LIN {X 0,Y 411.273,Z 176.254,A -85,B 0,C 180,E1 -10451.833,E2 -10451.833} C_VEL
LIN {X 0,Y 411.231,Z 176.261,A -85,B 0,C 180,E1 -10454.854,E2 -10454.854} C_VEL
LIN {X 0,Y 411.22,Z 176.261,A -85,B 0,C 180,E1 -10457.916,E2 -10457.916} C_VEL
LIN {X 0,Y 411.208,Z 176.265,A -85,B 0,C 180,E1 -10461.033,E2 -10461.033} C_VEL
LIN {X 0,Y 411.202,Z 176.262,A -85,B 0,C 180,E1 -10464.217,E2 -10464.217} C_VEL
LIN {X 0,Y 411.232,Z 176.258,A -85,B 0,C 180,E1 -10467.48,E2 -10467.48} C_VEL
LIN {X 0,Y 411.171,Z 176.269,A -85,B 0,C 180,E1 -10470.849,E2 -10470.849} C_VEL
LIN {X 0,Y 411.181,Z 176.268,A -85,B 0,C 180,E1 -10474.336,E2 -10474.336} C_VEL
LIN {X 0,Y 411.182,Z 176.266,A -85,B 0,C 180,E1 -10477.975,E2 -10477.975} C_VEL
LIN {X 0,Y 411.189,Z 176.264,A -85,B 0,C 180,E1 -10481.238,E2 -10481.238} C_VEL
LIN {X 0,Y 411.214,Z 176.264,A -85,B 0,C 180,E1 -10484.485,E2 -10484.485} C_VEL
LIN {X 0,Y 411.208,Z 176.268,A -85,B 0,C 180,E1 -10487.3,E2 -10487.3} C_VEL
LIN {X 0,Y 411.201,Z 176.348,A -85,B 0,C 180,E1 -10489.503,E2 -10489.503} C_VEL
LIN {X 0,Y 411.973,Z 180.687,A -85,B 0,C 180,E1 -10492.115,E2 -10492.115} C_VEL
LIN {X 0,Y 412.375,Z 185.022,A -85,B 0,C 180,E1 -10494.592,E2 -10494.592} C_VEL
LIN {X 0,Y 411.962,Z 191.551,A -85,B 0,C 180,E1 -10498.075,E2 -10498.075} C_VEL
LIN {X 0,Y 411.48,Z 198.091,A -85,B 0,C 180,E1 -10501.433,E2 -10501.433} C_VEL
LIN {X 0,Y 411.07,Z 205.195,A -85,B 0,C 180,E1 -10504.977,E2 -10504.977} C_VEL
LIN {X 0,Y 410.743,Z 212.225,A -85,B 0,C 180,E1 -10508.418,E2 -10508.418} C_VEL
LIN {X 0,Y 410.41,Z 219.753,A -85,B 0,C 180,E1 -10512.049,E2 -10512.049} C_VEL
LIN {X 0,Y 410.348,Z 220.824,A -85,B 0,C 180,E1 -10512.562,E2 -10512.562} C_VEL
LIN {X 0,Y 412.666,Z 234.125,A -85,B 0,C 180,E1 -10513.061,E2 -10513.061} C_VEL
LIN {X 0,Y 414.357,Z 246.561,A -85,B 0,C 180,E1 -10513.709,E2 -10513.709} C_VEL
LIN {X 0,Y 414.471,Z 252.147,A -85,B 0,C 180,E1 -10514.042,E2 -10514.042} C_VEL
LIN {X 0,Y 413.707,Z 263.943,A -85,B 0,C 180,E1 -10514.861,E2 -10514.861} C_VEL
LIN {X 0,Y 412.966,Z 274.206,A -85,B 0,C 180,E1 -10515.766,E2 -10515.766} C_VEL
LIN {X 0,Y 412.217,Z 284.881,A -85,B 0,C 180,E1 -10516.946,E2 -10516.946} C_VEL
LIN {X 0,Y 411.604,Z 293.906,A -85,B 0,C 180,E1 -10518.178,E2 -10518.178} C_VEL
LIN {X 0,Y 410.954,Z 302.716,A -85,B 0,C 180,E1 -10519.657,E2 -10519.657} C_VEL
LIN {X 0,Y 410.528,Z 309.753,A -85,B 0,C 180,E1 -10521.138,E2 -10521.138} C_VEL
LIN {X 0,Y 410.19,Z 315.381,A -85,B 0,C 180,E1 -10522.618,E2 -10522.618} C_VEL
LIN {X 0,Y 410.035,Z 319.809,A -85,B 0,C 180,E1 -10524.098,E2 -10524.098} C_VEL
LIN {X 0,Y 410.019,Z 322.149,A -85,B 0,C 180,E1 -10525.085,E2 -10525.085} C_VEL
LIN {X 0,Y 409.932,Z 324.056,A -85,B 0,C 180,E1 -10526.069,E2 -10526.069} C_VEL
LIN {X 0,Y 409.926,Z 325.518,A -85,B 0,C 180,E1 -10527.053,E2 -10527.053} C_VEL
LIN {X 0,Y 409.966,Z 326.551,A -85,B 0,C 180,E1 -10528.036,E2 -10528.036} C_VEL
LIN {X 0,Y 409.927,Z 327.448,A -85,B 0,C 180,E1 -10530.001,E2 -10530.001} C_VEL
LIN {X 0,Y 409.935,Z 327.293,A -85,B 0,C 180,E1 -10530.983,E2 -10530.983} C_VEL
LIN {X 0,Y 409.966,Z 326.72,A -85,B 0,C 180,E1 -10531.965,E2 -10531.965} C_VEL
LIN {X 0,Y 409.931,Z 324.402,A -85,B 0,C 180,E1 -10533.933,E2 -10533.933} C_VEL
LIN {X 0,Y 410.018,Z 321.536,A -85,B 0,C 180,E1 -10535.41,E2 -10535.41} C_VEL
LIN {X 0,Y 410.168,Z 317.645,A -85,B 0,C 180,E1 -10536.889,E2 -10536.889} C_VEL
LIN {X 0,Y 410.421,Z 312.629,A -85,B 0,C 180,E1 -10538.369,E2 -10538.369} C_VEL
LIN {X 0,Y 410.84,Z 306.335,A -85,B 0,C 180,E1 -10539.85,E2 -10539.85} C_VEL
LIN {X 0,Y 411.402,Z 298.458,A -85,B 0,C 180,E1 -10541.33,E2 -10541.33} C_VEL
LIN {X 0,Y 412.128,Z 290.44,A -85,B 0,C 180,E1 -10542.558,E2 -10542.558} C_VEL
LIN {X 0,Y 412.802,Z 280.664,A -85,B 0,C 180,E1 -10543.789,E2 -10543.789} C_VEL
LIN {X 0,Y 413.655,Z 269.786,A -85,B 0,C 180,E1 -10544.89,E2 -10544.89} C_VEL
LIN {X 0,Y 414.435,Z 259.142,A -85,B 0,C 180,E1 -10545.743,E2 -10545.743} C_VEL
LIN {X 0,Y 414.947,Z 248.593,A -85,B 0,C 180,E1 -10546.417,E2 -10546.417} C_VEL
LIN {X 0,Y 413.347,Z 236.158,A -85,B 0,C 180,E1 -10547.103,E2 -10547.103} C_VEL
LIN {X 0,Y 410.794,Z 222.945,A -85,B 0,C 180,E1 -10547.664,E2 -10547.664} C_VEL
LIN {X 0,Y 410.406,Z 220.684,A -85,B 0,C 180,E1 -10547.759,E2 -10547.759} C_VEL
LIN {X 0,Y 410.738,Z 213.884,A -85,B 0,C 180,E1 -10551.058,E2 -10551.058} C_VEL
LIN {X 0,Y 411.04,Z 207.48,A -85,B 0,C 180,E1 -10554.226,E2 -10554.226} C_VEL
LIN {X 0,Y 411.432,Z 201.028,A -85,B 0,C 180,E1 -10557.464,E2 -10557.464} C_VEL
LIN {X 0,Y 411.887,Z 194.581,A -85,B 0,C 180,E1 -10560.788,E2 -10560.788} C_VEL
LIN {X 0,Y 412.246,Z 189.772,A -85,B 0,C 180,E1 -10563.347,E2 -10563.347} C_VEL
LIN {X 0,Y 412.463,Z 184.976,A -85,B 0,C 180,E1 -10566.002,E2 -10566.002} C_VEL
LIN {X 0,Y 412.038,Z 181.046,A -85,B 0,C 180,E1 -10568.316,E2 -10568.316} C_VEL
LIN {X 0,Y 411.221,Z 176.262,A -85,B 0,C 180,E1 -10571.317,E2 -10571.317} C_VEL
LIN {X 0,Y 411.217,Z 176.263,A -85,B 0,C 180,E1 -10574.482,E2 -10574.482} C_VEL
LIN {X 0,Y 411.163,Z 176.268,A -85,B 0,C 180,E1 -10578.193,E2 -10578.193} C_VEL
LIN {X 0,Y 411.193,Z 176.264,A -85,B 0,C 180,E1 -10580.773,E2 -10580.773} C_VEL
LIN {X 0,Y 411.181,Z 176.264,A -85,B 0,C 180,E1 -10584.47,E2 -10584.47} C_VEL
LIN {X 0,Y 411.19,Z 176.265,A -85,B 0,C 180,E1 -10586.872,E2 -10586.872} C_VEL
LIN {X 0,Y 411.196,Z 176.264,A -85,B 0,C 180,E1 -10590.647,E2 -10590.647} C_VEL
LIN {X 0,Y 411.218,Z 176.261,A -85,B 0,C 180,E1 -10593.618,E2 -10593.618} C_VEL
LIN {X 0,Y 411.236,Z 176.259,A -85,B 0,C 180,E1 -10597.339,E2 -10597.339} C_VEL
LIN {X 0,Y 411.244,Z 176.256,A -85,B 0,C 180,E1 -10600.03,E2 -10600.03} C_VEL
LIN {X 0,Y 411.242,Z 176.26,A -85,B 0,C 180,E1 -10603.13,E2 -10603.13} C_VEL
LIN {X 0,Y 411.289,Z 176.255,A -85,B 0,C 180,E1 -10606.891,E2 -10606.891} C_VEL
LIN {X 0,Y 411.288,Z 176.253,A -85,B 0,C 180,E1 -10610.161,E2 -10610.161} C_VEL
LIN {X 0,Y 411.457,Z 176.23,A -85,B 0,C 180,E1 -10613.133,E2 -10613.133} C_VEL
LIN {X 0,Y 411.296,Z 176.251,A -85,B 0,C 180,E1 -10615.099,E2 -10615.099} C_VEL
LIN {X 0,Y 411.484,Z 176.231,A -85,B 0,C 180,E1 -10618.043,E2 -10618.043} C_VEL
LIN {X 0,Y 411.611,Z 176.214,A -85,B 0,C 180,E1 -10620,E2 -10620} C_VEL
LIN {X 0,Y 411.451,Z 176.23,A -85,B 0,C 180,E1 -10622.938,E2 -10622.938} C_VEL
LIN {X 0,Y 411.431,Z 176.233,A -85,B 0,C 180,E1 -10626.604,E2 -10626.604} C_VEL
LIN {X 0,Y 411.268,Z 176.258,A -85,B 0,C 180,E1 -10629.84,E2 -10629.84} C_VEL
LIN {X 0,Y 411.282,Z 176.253,A -85,B 0,C 180,E1 -10633.104,E2 -10633.104} C_VEL
LIN {X 0,Y 411.281,Z 176.251,A -85,B 0,C 180,E1 -10636.888,E2 -10636.888} C_VEL
LIN {X 0,Y 411.21,Z 176.263,A -85,B 0,C 180,E1 -10639.988,E2 -10639.988} C_VEL
LIN {X 0,Y 411.183,Z 176.268,A -85,B 0,C 180,E1 -10643.149,E2 -10643.149} C_VEL
LIN {X 0,Y 411.219,Z 176.259,A -85,B 0,C 180,E1 -10646.383,E2 -10646.383} C_VEL
LIN {X 0,Y 411.193,Z 176.264,A -85,B 0,C 180,E1 -10649.714,E2 -10649.714} C_VEL
LIN {X 0,Y 411.191,Z 176.267,A -85,B 0,C 180,E1 -10653.158,E2 -10653.158} C_VEL
LIN {X 0,Y 411.178,Z 176.267,A -85,B 0,C 180,E1 -10656.554,E2 -10656.554} C_VEL
LIN {X 0,Y 411.196,Z 176.262,A -85,B 0,C 180,E1 -10659.729,E2 -10659.729} C_VEL
LIN {X 0,Y 411.162,Z 176.269,A -85,B 0,C 180,E1 -10663.136,E2 -10663.136} C_VEL
LIN {X 0,Y 411.159,Z 176.267,A -85,B 0,C 180,E1 -10665.883,E2 -10665.883} C_VEL
LIN {X 0,Y 411.154,Z 176.272,A -85,B 0,C 180,E1 -10668.774,E2 -10668.774} C_VEL
LIN {X 0,Y 411.093,Z 176.295,A -85,B 0,C 180,E1 -10671.852,E2 -10671.852} C_VEL
LIN {X 0,Y 411.092,Z 179.421,A -85,B 0,C 180,E1 -10674.463,E2 -10674.463} C_VEL
LIN {X 0,Y 410.927,Z 183.802,A -85,B 0,C 180,E1 -10677.984,E2 -10677.984} C_VEL
LIN {X 0,Y 410.72,Z 188.143,A -85,B 0,C 180,E1 -10681.374,E2 -10681.374} C_VEL
LIN {X 0,Y 410.555,Z 192.532,A -85,B 0,C 180,E1 -10684.663,E2 -10684.663} C_VEL
LIN {X 0,Y 410.421,Z 196.937,A -85,B 0,C 180,E1 -10687.87,E2 -10687.87} C_VEL
LIN {X 0,Y 410.363,Z 200.38,A -85,B 0,C 180,E1 -10690.327,E2 -10690.327} C_VEL
LIN {X 0,Y 413.785,Z 215.04,A -85,B 0,C 180,E1 -10690.995,E2 -10690.995} C_VEL
LIN {X 0,Y 415.59,Z 225.146,A -85,B 0,C 180,E1 -10691.579,E2 -10691.579} C_VEL
LIN {X 0,Y 414.916,Z 237.745,A -85,B 0,C 180,E1 -10692.376,E2 -10692.376} C_VEL
LIN {X 0,Y 414.043,Z 249.487,A -85,B 0,C 180,E1 -10693.356,E2 -10693.356} C_VEL
LIN {X 0,Y 413.36,Z 258.933,A -85,B 0,C 180,E1 -10694.342,E2 -10694.342} C_VEL
LIN {X 0,Y 412.494,Z 269.466,A -85,B 0,C 180,E1 -10695.697,E2 -10695.697} C_VEL
LIN {X 0,Y 411.837,Z 277.292,A -85,B 0,C 180,E1 -10696.949,E2 -10696.949} C_VEL
LIN {X 0,Y 411.318,Z 284.751,A -85,B 0,C 180,E1 -10698.418,E2 -10698.418} C_VEL
LIN {X 0,Y 410.81,Z 289.915,A -85,B 0,C 180,E1 -10699.652,E2 -10699.652} C_VEL
LIN {X 0,Y 410.499,Z 294.904,A -85,B 0,C 180,E1 -10701.136,E2 -10701.136} C_VEL
LIN {X 0,Y 410.23,Z 298.768,A -85,B 0,C 180,E1 -10702.618,E2 -10702.618} C_VEL
LIN {X 0,Y 410.073,Z 301.606,A -85,B 0,C 180,E1 -10704.098,E2 -10704.098} C_VEL
LIN {X 0,Y 410.043,Z 302.944,A -85,B 0,C 180,E1 -10705.084,E2 -10705.084} C_VEL
LIN {X 0,Y 409.969,Z 304.457,A -85,B 0,C 180,E1 -10707.052,E2 -10707.052} C_VEL
LIN {X 0,Y 410.003,Z 304.609,A -85,B 0,C 180,E1 -10708.035,E2 -10708.035} C_VEL
LIN {X 0,Y 409.931,Z 303.724,A -85,B 0,C 180,E1 -10709.999,E2 -10709.999} C_VEL
LIN {X 0,Y 409.97,Z 302.708,A -85,B 0,C 180,E1 -10710.982,E2 -10710.982} C_VEL
LIN {X 0,Y 410.076,Z 301.27,A -85,B 0,C 180,E1 -10711.963,E2 -10711.963} C_VEL
LIN {X 0,Y 410.309,Z 298.319,A -85,B 0,C 180,E1 -10713.436,E2 -10713.436} C_VEL
LIN {X 0,Y 410.422,Z 294.338,A -85,B 0,C 180,E1 -10714.911,E2 -10714.911} C_VEL
LIN {X 0,Y 410.865,Z 288.202,A -85,B 0,C 180,E1 -10716.629,E2 -10716.629} C_VEL
LIN {X 0,Y 411.324,Z 281.524,A -85,B 0,C 180,E1 -10718.102,E2 -10718.102} C_VEL
LIN {X 0,Y 411.935,Z 273.234,A -85,B 0,C 180,E1 -10719.574,E2 -10719.574} C_VEL
LIN {X 0,Y 412.14,Z 271.122,A -85,B 0,C 180,E1 -10719.894,E2 -10719.894} C_VEL
LIN {X 0,Y 411.831,Z 267.118,A -85,B 0,C 180,E1 -10720.493,E2 -10720.493} C_VEL
LIN {X 0,Y 409.616,Z 260.349,A -85,B 0,C 180,E1 -10721.45,E2 -10721.45} C_VEL
LIN {X 0,Y 407.273,Z 253.153,A -85,B 0,C 180,E1 -10722.35,E2 -10722.35} C_VEL
LIN {X 0,Y 406.767,Z 248.372,A -85,B 0,C 180,E1 -10722.849,E2 -10722.849} C_VEL
LIN {X 0,Y 407.614,Z 237.96,A -85,B 0,C 180,E1 -10723.712,E2 -10723.712} C_VEL
LIN {X 0,Y 408.173,Z 227.39,A -85,B 0,C 180,E1 -10724.411,E2 -10724.411} C_VEL
LIN {X 0,Y 408.052,Z 223.747,A -85,B 0,C 180,E1 -10724.624,E2 -10724.624} C_VEL
LIN {X 0,Y 405.676,Z 211.271,A -85,B 0,C 180,E1 -10725.307,E2 -10725.307} C_VEL
LIN {X 0,Y 403.286,Z 200.508,A -85,B 0,C 180,E1 -10725.767,E2 -10725.767} C_VEL
LIN {X 0,Y 403.368,Z 195.566,A -85,B 0,C 180,E1 -10729.33,E2 -10729.33} C_VEL
LIN {X 0,Y 403.532,Z 191.072,A -85,B 0,C 180,E1 -10732.621,E2 -10732.621} C_VEL
LIN {X 0,Y 403.664,Z 186.904,A -85,B 0,C 180,E1 -10735.799,E2 -10735.799} C_VEL
LIN {X 0,Y 403.861,Z 182.638,A -85,B 0,C 180,E1 -10739.157,E2 -10739.157} C_VEL
LIN {X 0,Y 403.988,Z 179.68,A -85,B 0,C 180,E1 -10741.522,E2 -10741.522} C_VEL
LIN {X 0,Y 403.986,Z 177.43,A -85,B 0,C 180,E1 -10743.379,E2 -10743.379} C_VEL
LIN {X 0,Y 404.088,Z 177.151,A -85,B 0,C 180,E1 -10745.17,E2 -10745.17} C_VEL
LIN {X 0,Y 404.136,Z 177.142,A -85,B 0,C 180,E1 -10748.504,E2 -10748.504} C_VEL
LIN {X 0,Y 404.11,Z 177.149,A -85,B 0,C 180,E1 -10751.597,E2 -10751.597} C_VEL
LIN {X 0,Y 404.141,Z 177.142,A -85,B 0,C 180,E1 -10754.521,E2 -10754.521} C_VEL
LIN {X 0,Y 404.189,Z 177.139,A -85,B 0,C 180,E1 -10757.302,E2 -10757.302} C_VEL
LIN {X 0,Y 404.15,Z 177.14,A -85,B 0,C 180,E1 -10759.953,E2 -10759.953} C_VEL
LIN {X 0,Y 404.116,Z 177.148,A -85,B 0,C 180,E1 -10763.122,E2 -10763.122} C_VEL
LIN {X 0,Y 404.122,Z 177.145,A -85,B 0,C 180,E1 -10766.185,E2 -10766.185} C_VEL
LIN {X 0,Y 404.128,Z 177.143,A -85,B 0,C 180,E1 -10769.713,E2 -10769.713} C_VEL
LIN {X 0,Y 404.17,Z 177.139,A -85,B 0,C 180,E1 -10773.121,E2 -10773.121} C_VEL
LIN {X 0,Y 404.154,Z 177.144,A -85,B 0,C 180,E1 -10776.424,E2 -10776.424} C_VEL
LIN {X 0,Y 404.198,Z 177.136,A -85,B 0,C 180,E1 -10779.859,E2 -10779.859} C_VEL
LIN {X 0,Y 404.188,Z 177.137,A -85,B 0,C 180,E1 -10782.99,E2 -10782.99} C_VEL
LIN {X 0,Y 404.197,Z 177.138,A -85,B 0,C 180,E1 -10785.911,E2 -10785.911} C_VEL
LIN {X 0,Y 404.254,Z 177.127,A -85,B 0,C 180,E1 -10788.975,E2 -10788.975} C_VEL
LIN {X 0,Y 404.402,Z 177.113,A -85,B 0,C 180,E1 -10792.097,E2 -10792.097} C_VEL
LIN {X 0,Y 404.418,Z 177.111,A -85,B 0,C 180,E1 -10794.015,E2 -10794.015} C_VEL
LIN {X 0,Y 404.447,Z 177.107,A -85,B 0,C 180,E1 -10798.008,E2 -10798.008} C_VEL
LIN {X 0,Y 404.574,Z 177.091,A -85,B 0,C 180,E1 -10800,E2 -10800} C_VEL
LIN {X 0,Y 404.4,Z 177.11,A -85,B 0,C 180,E1 -10802.988,E2 -10802.988} C_VEL
LIN {X 0,Y 404.409,Z 177.11,A -85,B 0,C 180,E1 -10805.985,E2 -10805.985} C_VEL
LIN {X 0,Y 404.289,Z 177.124,A -85,B 0,C 180,E1 -10809.001,E2 -10809.001} C_VEL
LIN {X 0,Y 404.242,Z 177.129,A -85,B 0,C 180,E1 -10812.042,E2 -10812.042} C_VEL
LIN {X 0,Y 404.176,Z 177.142,A -85,B 0,C 180,E1 -10815.119,E2 -10815.119} C_VEL
LIN {X 0,Y 404.181,Z 177.137,A -85,B 0,C 180,E1 -10818.239,E2 -10818.239} C_VEL
LIN {X 0,Y 404.164,Z 177.142,A -85,B 0,C 180,E1 -10821.418,E2 -10821.418} C_VEL
LIN {X 0,Y 404.151,Z 177.143,A -85,B 0,C 180,E1 -10824.667,E2 -10824.667} C_VEL
LIN {X 0,Y 404.17,Z 177.137,A -85,B 0,C 180,E1 -10828.001,E2 -10828.001} C_VEL
LIN {X 0,Y 404.116,Z 177.145,A -85,B 0,C 180,E1 -10831.561,E2 -10831.561} C_VEL
LIN {X 0,Y 404.161,Z 177.142,A -85,B 0,C 180,E1 -10835.018,E2 -10835.018} C_VEL
LIN {X 0,Y 404.142,Z 177.145,A -85,B 0,C 180,E1 -10838.758,E2 -10838.758} C_VEL
LIN {X 0,Y 404.171,Z 177.138,A -85,B 0,C 180,E1 -10841.613,E2 -10841.613} C_VEL
LIN {X 0,Y 404.179,Z 177.14,A -85,B 0,C 180,E1 -10844.532,E2 -10844.532} C_VEL
LIN {X 0,Y 404.187,Z 177.143,A -85,B 0,C 180,E1 -10847.307,E2 -10847.307} C_VEL
LIN {X 0,Y 404.187,Z 177.286,A -85,B 0,C 180,E1 -10849.309,E2 -10849.309} C_VEL
LIN {X 0,Y 404.938,Z 181.679,A -85,B 0,C 180,E1 -10852.001,E2 -10852.001} C_VEL
LIN {X 0,Y 405.354,Z 186.104,A -85,B 0,C 180,E1 -10854.576,E2 -10854.576} C_VEL
LIN {X 0,Y 404.913,Z 192.898,A -85,B 0,C 180,E1 -10858.264,E2 -10858.264} C_VEL
LIN {X 0,Y 404.428,Z 199.01,A -85,B 0,C 180,E1 -10861.456,E2 -10861.456} C_VEL
LIN {X 0,Y 404.048,Z 205.484,A -85,B 0,C 180,E1 -10864.754,E2 -10864.754} C_VEL
LIN {X 0,Y 403.652,Z 213.104,A -85,B 0,C 180,E1 -10868.556,E2 -10868.556} C_VEL
LIN {X 0,Y 403.301,Z 220.736,A -85,B 0,C 180,E1 -10872.265,E2 -10872.265} C_VEL
LIN {X 0,Y 405.694,Z 234.188,A -85,B 0,C 180,E1 -10872.787,E2 -10872.787} C_VEL
LIN {X 0,Y 407.406,Z 246.932,A -85,B 0,C 180,E1 -10873.47,E2 -10873.47} C_VEL
LIN {X 0,Y 407.615,Z 252.022,A -85,B 0,C 180,E1 -10873.784,E2 -10873.784} C_VEL
LIN {X 0,Y 406.827,Z 263.573,A -85,B 0,C 180,E1 -10874.599,E2 -10874.599} C_VEL
LIN {X 0,Y 405.996,Z 274.629,A -85,B 0,C 180,E1 -10875.593,E2 -10875.593} C_VEL
LIN {X 0,Y 405.276,Z 284.759,A -85,B 0,C 180,E1 -10876.742,E2 -10876.742} C_VEL
LIN {X 0,Y 404.622,Z 293.619,A -85,B 0,C 180,E1 -10877.971,E2 -10877.971} C_VEL
LIN {X 0,Y 403.918,Z 302.445,A -85,B 0,C 180,E1 -10879.475,E2 -10879.475} C_VEL
LIN {X 0,Y 403.483,Z 309.501,A -85,B 0,C 180,E1 -10880.982,E2 -10880.982} C_VEL
LIN {X 0,Y 403.137,Z 315.141,A -85,B 0,C 180,E1 -10882.488,E2 -10882.488} C_VEL
LIN {X 0,Y 402.966,Z 319.578,A -85,B 0,C 180,E1 -10883.994,E2 -10883.994} C_VEL
LIN {X 0,Y 402.932,Z 321.923,A -85,B 0,C 180,E1 -10884.998,E2 -10884.998} C_VEL
LIN {X 0,Y 402.852,Z 323.835,A -85,B 0,C 180,E1 -10885.999,E2 -10885.999} C_VEL
LIN {X 0,Y 402.825,Z 325.305,A -85,B 0,C 180,E1 -10887.001,E2 -10887.001} C_VEL
LIN {X 0,Y 402.864,Z 326.342,A -85,B 0,C 180,E1 -10888.001,E2 -10888.001} C_VEL
LIN {X 0,Y 402.862,Z 326.989,A -85,B 0,C 180,E1 -10889.001,E2 -10889.001} C_VEL
LIN {X 0,Y 402.851,Z 327.249,A -85,B 0,C 180,E1 -10890.001,E2 -10890.001} C_VEL
LIN {X 0,Y 402.862,Z 327.103,A -85,B 0,C 180,E1 -10891,E2 -10891} C_VEL
LIN {X 0,Y 402.864,Z 326.533,A -85,B 0,C 180,E1 -10892,E2 -10892} C_VEL
LIN {X 0,Y 402.852,Z 324.223,A -85,B 0,C 180,E1 -10894.002,E2 -10894.002} C_VEL
LIN {X 0,Y 402.916,Z 321.366,A -85,B 0,C 180,E1 -10895.505,E2 -10895.505} C_VEL
LIN {X 0,Y 403.082,Z 317.484,A -85,B 0,C 180,E1 -10897.011,E2 -10897.011} C_VEL
LIN {X 0,Y 403.363,Z 312.478,A -85,B 0,C 180,E1 -10898.517,E2 -10898.517} C_VEL
LIN {X 0,Y 403.829,Z 306.197,A -85,B 0,C 180,E1 -10900.022,E2 -10900.022} C_VEL
LIN {X 0,Y 404.417,Z 298.339,A -85,B 0,C 180,E1 -10901.528,E2 -10901.528} C_VEL
LIN {X 0,Y 405.173,Z 290.338,A -85,B 0,C 180,E1 -10902.777,E2 -10902.777} C_VEL
LIN {X 0,Y 405.871,Z 280.581,A -85,B 0,C 180,E1 -10904.029,E2 -10904.029} C_VEL
LIN {X 0,Y 406.791,Z 269.735,A -85,B 0,C 180,E1 -10905.147,E2 -10905.147} C_VEL
LIN {X 0,Y 407.604,Z 259.135,A -85,B 0,C 180,E1 -10906.014,E2 -10906.014} C_VEL
LIN {X 0,Y 408.152,Z 249.946,A -85,B 0,C 180,E1 -10906.621,E2 -10906.621} C_VEL
LIN {X 0,Y 406.835,Z 238.963,A -85,B 0,C 180,E1 -10907.269,E2 -10907.269} C_VEL
LIN {X 0,Y 404.358,Z 225.626,A -85,B 0,C 180,E1 -10907.886,E2 -10907.886} C_VEL
LIN {X 0,Y 403.357,Z 220.523,A -85,B 0,C 180,E1 -10908.08,E2 -10908.08} C_VEL
LIN {X 0,Y 403.693,Z 213.717,A -85,B 0,C 180,E1 -10911.443,E2 -10911.443} C_VEL
LIN {X 0,Y 404.044,Z 207.354,A -85,B 0,C 180,E1 -10914.673,E2 -10914.673} C_VEL
LIN {X 0,Y 404.551,Z 199.834,A -85,B 0,C 180,E1 -10918.536,E2 -10918.536} C_VEL
LIN {X 0,Y 404.941,Z 194.473,A -85,B 0,C 180,E1 -10921.375,E2 -10921.375} C_VEL
LIN {X 0,Y 405.393,Z 189.145,A -85,B 0,C 180,E1 -10924.291,E2 -10924.291} C_VEL
LIN {X 0,Y 405.465,Z 185.958,A -85,B 0,C 180,E1 -10926.107,E2 -10926.107} C_VEL
LIN {X 0,Y 404.946,Z 181.716,A -85,B 0,C 180,E1 -10928.665,E2 -10928.665} C_VEL
LIN {X 0,Y 404.198,Z 177.138,A -85,B 0,C 180,E1 -10931.612,E2 -10931.612} C_VEL
LIN {X 0,Y 404.181,Z 177.139,A -85,B 0,C 180,E1 -10934.527,E2 -10934.527} C_VEL
LIN {X 0,Y 404.123,Z 177.149,A -85,B 0,C 180,E1 -10937.294,E2 -10937.294} C_VEL
LIN {X 0,Y 404.14,Z 177.144,A -85,B 0,C 180,E1 -10939.952,E2 -10939.952} C_VEL
LIN {X 0,Y 404.12,Z 177.147,A -85,B 0,C 180,E1 -10943.124,E2 -10943.124} C_VEL
LIN {X 0,Y 404.128,Z 177.142,A -85,B 0,C 180,E1 -10946.186,E2 -10946.186} C_VEL
LIN {X 0,Y 404.127,Z 177.145,A -85,B 0,C 180,E1 -10949.713,E2 -10949.713} C_VEL
LIN {X 0,Y 404.176,Z 177.141,A -85,B 0,C 180,E1 -10953.122,E2 -10953.122} C_VEL
LIN {X 0,Y 404.16,Z 177.14,A -85,B 0,C 180,E1 -10956.425,E2 -10956.425} C_VEL
LIN {X 0,Y 404.205,Z 177.133,A -85,B 0,C 180,E1 -10959.86,E2 -10959.86} C_VEL
LIN {X 0,Y 404.197,Z 177.138,A -85,B 0,C 180,E1 -10962.991,E2 -10962.991} C_VEL
LIN {X 0,Y 404.244,Z 177.133,A -85,B 0,C 180,E1 -10966.788,E2 -10966.788} C_VEL
LIN {X 0,Y 404.25,Z 177.128,A -85,B 0,C 180,E1 -10969.988,E2 -10969.988} C_VEL
LIN {X 0,Y 404.418,Z 177.108,A -85,B 0,C 180,E1 -10973.013,E2 -10973.013} C_VEL
LIN {X 0,Y 404.269,Z 177.126,A -85,B 0,C 180,E1 -10975.014,E2 -10975.014} C_VEL
LIN {X 0,Y 404.453,Z 177.106,A -85,B 0,C 180,E1 -10978.009,E2 -10978.009} C_VEL
LIN {X 0,Y 404.581,Z 177.09,A -85,B 0,C 180,E1 -10980,E2 -10980} C_VEL
LIN {X 0,Y 404.409,Z 177.107,A -85,B 0,C 180,E1 -10982.989,E2 -10982.989} C_VEL
LIN {X 0,Y 404.377,Z 177.112,A -85,B 0,C 180,E1 -10986.6,E2 -10986.6} C_VEL
LIN {X 0,Y 404.266,Z 177.126,A -85,B 0,C 180,E1 -10989.002,E2 -10989.002} C_VEL
LIN {X 0,Y 404.232,Z 177.134,A -85,B 0,C 180,E1 -10992.043,E2 -10992.043} C_VEL
LIN {X 0,Y 404.19,Z 177.136,A -85,B 0,C 180,E1 -10995.119,E2 -10995.119} C_VEL
LIN {X 0,Y 404.194,Z 177.135,A -85,B 0,C 180,E1 -10998.239,E2 -10998.239} C_VEL
LIN {X 0,Y 404.118,Z 177.149,A -85,B 0,C 180,E1 -11001.421,E2 -11001.421} C_VEL
LIN {X 0,Y 404.158,Z 177.14,A -85,B 0,C 180,E1 -11004.667,E2 -11004.667} C_VEL
LIN {X 0,Y 404.18,Z 177.136,A -85,B 0,C 180,E1 -11008.001,E2 -11008.001} C_VEL
LIN {X 0,Y 404.126,Z 177.146,A -85,B 0,C 180,E1 -11011.56,E2 -11011.56} C_VEL
LIN {X 0,Y 404.169,Z 177.142,A -85,B 0,C 180,E1 -11015.018,E2 -11015.018} C_VEL
LIN {X 0,Y 404.138,Z 177.145,A -85,B 0,C 180,E1 -11018.759,E2 -11018.759} C_VEL
LIN {X 0,Y 404.111,Z 177.144,A -85,B 0,C 180,E1 -11021.601,E2 -11021.601} C_VEL
LIN {X 0,Y 404.135,Z 177.146,A -85,B 0,C 180,E1 -11024.524,E2 -11024.524} C_VEL
LIN {X 0,Y 404.128,Z 177.144,A -85,B 0,C 180,E1 -11027.297,E2 -11027.297} C_VEL
LIN {X 0,Y 404.126,Z 177.144,A -85,B 0,C 180,E1 -11029.953,E2 -11029.953} C_VEL
LIN {X 0,Y 404.079,Z 177.155,A -85,B 0,C 180,E1 -11031.506,E2 -11031.506} C_VEL
LIN {X 0,Y 404.107,Z 179.531,A -85,B 0,C 180,E1 -11033.752,E2 -11033.752} C_VEL
LIN {X 0,Y 403.96,Z 183.003,A -85,B 0,C 180,E1 -11036.626,E2 -11036.626} C_VEL
LIN {X 0,Y 403.788,Z 186.816,A -85,B 0,C 180,E1 -11039.687,E2 -11039.687} C_VEL
LIN {X 0,Y 403.568,Z 191.19,A -85,B 0,C 180,E1 -11043.079,E2 -11043.079} C_VEL
LIN {X 0,Y 403.412,Z 195.616,A -85,B 0,C 180,E1 -11046.38,E2 -11046.38} C_VEL
LIN {X 0,Y 403.293,Z 200.581,A -85,B 0,C 180,E1 -11049.997,E2 -11049.997} C_VEL
LIN {X 0,Y 406.646,Z 214.4,A -85,B 0,C 180,E1 -11050.634,E2 -11050.634} C_VEL
LIN {X 0,Y 408.658,Z 224.962,A -85,B 0,C 180,E1 -11051.255,E2 -11051.255} C_VEL
LIN {X 0,Y 408.227,Z 235.887,A -85,B 0,C 180,E1 -11051.948,E2 -11051.948} C_VEL
LIN {X 0,Y 407.453,Z 246.785,A -85,B 0,C 180,E1 -11052.82,E2 -11052.82} C_VEL
LIN {X 0,Y 406.517,Z 257.883,A -85,B 0,C 180,E1 -11053.942,E2 -11053.942} C_VEL
LIN {X 0,Y 405.73,Z 267.745,A -85,B 0,C 180,E1 -11055.197,E2 -11055.197} C_VEL
LIN {X 0,Y 404.905,Z 276.606,A -85,B 0,C 180,E1 -11056.585,E2 -11056.585} C_VEL
LIN {X 0,Y 404.468,Z 283.728,A -85,B 0,C 180,E1 -11057.965,E2 -11057.965} C_VEL
LIN {X 0,Y 403.788,Z 290.037,A -85,B 0,C 180,E1 -11059.47,E2 -11059.47} C_VEL
LIN {X 0,Y 403.452,Z 295.043,A -85,B 0,C 180,E1 -11060.98,E2 -11060.98} C_VEL
LIN {X 0,Y 403.166,Z 298.921,A -85,B 0,C 180,E1 -11062.488,E2 -11062.488} C_VEL
LIN {X 0,Y 402.99,Z 301.774,A -85,B 0,C 180,E1 -11063.993,E2 -11063.993} C_VEL
LIN {X 0,Y 402.954,Z 303.118,A -85,B 0,C 180,E1 -11064.997,E2 -11064.997} C_VEL
LIN {X 0,Y 402.869,Z 304.645,A -85,B 0,C 180,E1 -11067,E2 -11067} C_VEL
LIN {X 0,Y 402.914,Z 304.81,A -85,B 0,C 180,E1 -11068,E2 -11068} C_VEL
LIN {X 0,Y 402.855,Z 303.938,A -85,B 0,C 180,E1 -11069.999,E2 -11069.999} C_VEL
LIN {X 0,Y 402.897,Z 302.929,A -85,B 0,C 180,E1 -11070.999,E2 -11070.999} C_VEL
LIN {X 0,Y 403.009,Z 301.505,A -85,B 0,C 180,E1 -11071.998,E2 -11071.998} C_VEL
LIN {X 0,Y 403.248,Z 298.565,A -85,B 0,C 180,E1 -11073.496,E2 -11073.496} C_VEL
LIN {X 0,Y 403.358,Z 294.6,A -85,B 0,C 180,E1 -11074.997,E2 -11074.997} C_VEL
LIN {X 0,Y 403.824,Z 288.484,A -85,B 0,C 180,E1 -11076.745,E2 -11076.745} C_VEL
LIN {X 0,Y 404.308,Z 281.825,A -85,B 0,C 180,E1 -11078.244,E2 -11078.244} C_VEL
LIN {X 0,Y 404.957,Z 273.561,A -85,B 0,C 180,E1 -11079.741,E2 -11079.741} C_VEL
LIN {X 0,Y 405.707,Z 265.046,A -85,B 0,C 180,E1 -11080.983,E2 -11080.983} C_VEL
LIN {X 0,Y 406.466,Z 254.553,A -85,B 0,C 180,E1 -11082.227,E2 -11082.227} C_VEL
LIN {X 0,Y 406.767,Z 248.372,A -85,B 0,C 180,E1 -11082.849,E2 -11082.849} C_VEL
LIN {X 0,Y 406.231,Z 245.152,A -85,B 0,C 180,E1 -11083.178,E2 -11083.178} C_VEL
LIN {X 0,Y 401.532,Z 234.763,A -85,B 0,C 180,E1 -11084.199,E2 -11084.199} C_VEL
LIN {X 0,Y 401.111,Z 231.243,A -85,B 0,C 180,E1 -11084.456,E2 -11084.456} C_VEL
LIN {X 0,Y 401.356,Z 225.73,A -85,B 0,C 180,E1 -11084.791,E2 -11084.791} C_VEL
LIN {X 0,Y 398.975,Z 212.913,A -85,B 0,C 180,E1 -11085.532,E2 -11085.532} C_VEL
LIN {X 0,Y 396.224,Z 200.698,A -85,B 0,C 180,E1 -11086.088,E2 -11086.088} C_VEL
LIN {X 0,Y 396.331,Z 195.393,A -85,B 0,C 180,E1 -11089.975,E2 -11089.975} C_VEL
LIN {X 0,Y 396.472,Z 191.389,A -85,B 0,C 180,E1 -11092.951,E2 -11092.951} C_VEL
LIN {X 0,Y 396.625,Z 187.098,A -85,B 0,C 180,E1 -11096.292,E2 -11096.292} C_VEL
LIN {X 0,Y 396.817,Z 182.702,A -85,B 0,C 180,E1 -11099.791,E2 -11099.791} C_VEL
LIN {X 0,Y 396.942,Z 179.925,A -85,B 0,C 180,E1 -11102.08,E2 -11102.08} C_VEL
LIN {X 0,Y 396.946,Z 178.047,A -85,B 0,C 180,E1 -11103.679,E2 -11103.679} C_VEL
LIN {X 0,Y 397.064,Z 178.026,A -85,B 0,C 180,E1 -11105.735,E2 -11105.735} C_VEL
LIN {X 0,Y 397.113,Z 178.018,A -85,B 0,C 180,E1 -11108.857,E2 -11108.857} C_VEL
LIN {X 0,Y 397.056,Z 178.024,A -85,B 0,C 180,E1 -11112.264,E2 -11112.264} C_VEL
LIN {X 0,Y 397.102,Z 178.022,A -85,B 0,C 180,E1 -11115.062,E2 -11115.062} C_VEL
LIN {X 0,Y 397.138,Z 178.013,A -85,B 0,C 180,E1 -11118.004,E2 -11118.004} C_VEL
LIN {X 0,Y 397.086,Z 178.02,A -85,B 0,C 180,E1 -11121.723,E2 -11121.723} C_VEL
LIN {X 0,Y 397.102,Z 178.019,A -85,B 0,C 180,E1 -11125.504,E2 -11125.504} C_VEL
LIN {X 0,Y 397.059,Z 178.026,A -85,B 0,C 180,E1 -11129.115,E2 -11129.115} C_VEL
LIN {X 0,Y 397.169,Z 178.014,A -85,B 0,C 180,E1 -11132.608,E2 -11132.608} C_VEL
LIN {X 0,Y 397.112,Z 178.017,A -85,B 0,C 180,E1 -11135.98,E2 -11135.98} C_VEL
LIN {X 0,Y 397.127,Z 178.015,A -85,B 0,C 180,E1 -11139.271,E2 -11139.271} C_VEL
LIN {X 0,Y 397.153,Z 178.014,A -85,B 0,C 180,E1 -11142.843,E2 -11142.843} C_VEL
LIN {X 0,Y 397.161,Z 178.012,A -85,B 0,C 180,E1 -11145.656,E2 -11145.656} C_VEL
LIN {X 0,Y 397.199,Z 178.007,A -85,B 0,C 180,E1 -11148.776,E2 -11148.776} C_VEL
LIN {X 0,Y 397.367,Z 177.991,A -85,B 0,C 180,E1 -11152.036,E2 -11152.036} C_VEL
LIN {X 0,Y 397.369,Z 177.99,A -85,B 0,C 180,E1 -11153.908,E2 -11153.908} C_VEL
LIN {X 0,Y 397.416,Z 177.983,A -85,B 0,C 180,E1 -11157.973,E2 -11157.973} C_VEL
LIN {X 0,Y 397.544,Z 177.967,A -85,B 0,C 180,E1 -11160,E2 -11160} C_VEL
LIN {X 0,Y 397.358,Z 177.987,A -85,B 0,C 180,E1 -11163.041,E2 -11163.041} C_VEL
LIN {X 0,Y 397.358,Z 177.987,A -85,B 0,C 180,E1 -11166.092,E2 -11166.092} C_VEL
LIN {X 0,Y 397.347,Z 177.988,A -85,B 0,C 180,E1 -11168.134,E2 -11168.134} C_VEL
LIN {X 0,Y 397.2,Z 178.005,A -85,B 0,C 180,E1 -11172.259,E2 -11172.259} C_VEL
LIN {X 0,Y 397.148,Z 178.016,A -85,B 0,C 180,E1 -11175.393,E2 -11175.393} C_VEL
LIN {X 0,Y 397.139,Z 178.015,A -85,B 0,C 180,E1 -11178.574,E2 -11178.574} C_VEL
LIN {X 0,Y 397.138,Z 178.014,A -85,B 0,C 180,E1 -11181.816,E2 -11181.816} C_VEL
LIN {X 0,Y 397.125,Z 178.016,A -85,B 0,C 180,E1 -11185.514,E2 -11185.514} C_VEL
LIN {X 0,Y 397.1,Z 178.021,A -85,B 0,C 180,E1 -11188.545,E2 -11188.545} C_VEL
LIN {X 0,Y 397.054,Z 178.025,A -85,B 0,C 180,E1 -11192.074,E2 -11192.074} C_VEL
LIN {X 0,Y 397.096,Z 178.019,A -85,B 0,C 180,E1 -11195.506,E2 -11195.506} C_VEL
LIN {X 0,Y 397.116,Z 178.019,A -85,B 0,C 180,E1 -11198.865,E2 -11198.865} C_VEL
LIN {X 0,Y 397.139,Z 178.017,A -85,B 0,C 180,E1 -11202.258,E2 -11202.258} C_VEL
LIN {X 0,Y 397.133,Z 178.015,A -85,B 0,C 180,E1 -11205.062,E2 -11205.062} C_VEL
LIN {X 0,Y 397.124,Z 178.025,A -85,B 0,C 180,E1 -11208.426,E2 -11208.426} C_VEL
LIN {X 0,Y 397.171,Z 178.223,A -85,B 0,C 180,E1 -11209.106,E2 -11209.106} C_VEL
LIN {X 0,Y 397.886,Z 182.555,A -85,B 0,C 180,E1 -11211.818,E2 -11211.818} C_VEL
LIN {X 0,Y 398.322,Z 186.896,A -85,B 0,C 180,E1 -11214.395,E2 -11214.395} C_VEL
LIN {X 0,Y 397.973,Z 192.319,A -85,B 0,C 180,E1 -11217.415,E2 -11217.415} C_VEL
LIN {X 0,Y 397.468,Z 198.829,A -85,B 0,C 180,E1 -11220.908,E2 -11220.908} C_VEL
LIN {X 0,Y 396.953,Z 206.419,A -85,B 0,C 180,E1 -11224.857,E2 -11224.857} C_VEL
LIN {X 0,Y 396.622,Z 212.899,A -85,B 0,C 180,E1 -11228.156,E2 -11228.156} C_VEL
LIN {X 0,Y 396.233,Z 220.369,A -85,B 0,C 180,E1 -11231.919,E2 -11231.919} C_VEL
LIN {X 0,Y 399.09,Z 236.875,A -85,B 0,C 180,E1 -11232.631,E2 -11232.631} C_VEL
LIN {X 0,Y 400.633,Z 248.851,A -85,B 0,C 180,E1 -11233.318,E2 -11233.318} C_VEL
LIN {X 0,Y 400.455,Z 256.52,A -85,B 0,C 180,E1 -11233.825,E2 -11233.825} C_VEL
LIN {X 0,Y 399.616,Z 267.642,A -85,B 0,C 180,E1 -11234.706,E2 -11234.706} C_VEL
LIN {X 0,Y 398.75,Z 278.457,A -85,B 0,C 180,E1 -11235.785,E2 -11235.785} C_VEL
LIN {X 0,Y 398.062,Z 288.131,A -85,B 0,C 180,E1 -11236.992,E2 -11236.992} C_VEL
LIN {X 0,Y 397.381,Z 296.499,A -85,B 0,C 180,E1 -11238.266,E2 -11238.266} C_VEL
LIN {X 0,Y 396.752,Z 304.686,A -85,B 0,C 180,E1 -11239.798,E2 -11239.798} C_VEL
LIN {X 0,Y 396.315,Z 311.276,A -85,B 0,C 180,E1 -11241.332,E2 -11241.332} C_VEL
LIN {X 0,Y 396.004,Z 316.523,A -85,B 0,C 180,E1 -11242.865,E2 -11242.865} C_VEL
LIN {X 0,Y 395.847,Z 320.026,A -85,B 0,C 180,E1 -11244.164,E2 -11244.164} C_VEL
LIN {X 0,Y 395.775,Z 323.613,A -85,B 0,C 180,E1 -11245.928,E2 -11245.928} C_VEL
LIN {X 0,Y 395.728,Z 325.092,A -85,B 0,C 180,E1 -11246.947,E2 -11246.947} C_VEL
LIN {X 0,Y 395.763,Z 326.133,A -85,B 0,C 180,E1 -11247.965,E2 -11247.965} C_VEL
LIN {X 0,Y 395.791,Z 326.785,A -85,B 0,C 180,E1 -11248.983,E2 -11248.983} C_VEL
LIN {X 0,Y 395.778,Z 327.05,A -85,B 0,C 180,E1 -11250.001,E2 -11250.001} C_VEL
LIN {X 0,Y 395.791,Z 326.911,A -85,B 0,C 180,E1 -11251.018,E2 -11251.018} C_VEL
LIN {X 0,Y 395.762,Z 326.345,A -85,B 0,C 180,E1 -11252.036,E2 -11252.036} C_VEL
LIN {X 0,Y 395.774,Z 324.045,A -85,B 0,C 180,E1 -11254.074,E2 -11254.074} C_VEL
LIN {X 0,Y 395.827,Z 320.767,A -85,B 0,C 180,E1 -11255.806,E2 -11255.806} C_VEL
LIN {X 0,Y 396.082,Z 315.785,A -85,B 0,C 180,E1 -11257.648,E2 -11257.648} C_VEL
LIN {X 0,Y 396.52,Z 309.365,A -85,B 0,C 180,E1 -11259.436,E2 -11259.436} C_VEL
LIN {X 0,Y 397.056,Z 302.363,A -85,B 0,C 180,E1 -11260.969,E2 -11260.969} C_VEL
LIN {X 0,Y 397.939,Z 293.605,A -85,B 0,C 180,E1 -11262.494,E2 -11262.494} C_VEL
LIN {X 0,Y 398.739,Z 283.499,A -85,B 0,C 180,E1 -11263.917,E2 -11263.917} C_VEL
LIN {X 0,Y 399.586,Z 273.821,A -85,B 0,C 180,E1 -11265.01,E2 -11265.01} C_VEL
LIN {X 0,Y 400.529,Z 262.352,A -85,B 0,C 180,E1 -11266.043,E2 -11266.043} C_VEL
LIN {X 0,Y 401.308,Z 252.184,A -85,B 0,C 180,E1 -11266.767,E2 -11266.767} C_VEL
LIN {X 0,Y 400.228,Z 241.487,A -85,B 0,C 180,E1 -11267.441,E2 -11267.441} C_VEL
LIN {X 0,Y 397.97,Z 228.461,A -85,B 0,C 180,E1 -11268.102,E2 -11268.102} C_VEL
LIN {X 0,Y 396.313,Z 220.291,A -85,B 0,C 180,E1 -11268.441,E2 -11268.441} C_VEL
LIN {X 0,Y 396.754,Z 212.535,A -85,B 0,C 180,E1 -11272.385,E2 -11272.385} C_VEL
LIN {X 0,Y 397.077,Z 206.549,A -85,B 0,C 180,E1 -11275.489,E2 -11275.489} C_VEL
LIN {X 0,Y 397.58,Z 199.723,A -85,B 0,C 180,E1 -11279.084,E2 -11279.084} C_VEL
LIN {X 0,Y 398.016,Z 194.245,A -85,B 0,C 180,E1 -11282.052,E2 -11282.052} C_VEL
LIN {X 0,Y 398.41,Z 189.054,A -85,B 0,C 180,E1 -11284.979,E2 -11284.979} C_VEL
LIN {X 0,Y 398.244,Z 184.951,A -85,B 0,C 180,E1 -11287.426,E2 -11287.426} C_VEL
LIN {X 0,Y 397.476,Z 180.104,A -85,B 0,C 180,E1 -11290.509,E2 -11290.509} C_VEL
LIN {X 0,Y 397.155,Z 178.017,A -85,B 0,C 180,E1 -11291.993,E2 -11291.993} C_VEL
LIN {X 0,Y 397.1,Z 178.02,A -85,B 0,C 180,E1 -11295.064,E2 -11295.064} C_VEL
LIN {X 0,Y 397.052,Z 178.026,A -85,B 0,C 180,E1 -11298.02,E2 -11298.02} C_VEL
LIN {X 0,Y 397.11,Z 178.02,A -85,B 0,C 180,E1 -11301.138,E2 -11301.138} C_VEL
LIN {X 0,Y 397.103,Z 178.017,A -85,B 0,C 180,E1 -11304.495,E2 -11304.495} C_VEL
LIN {X 0,Y 397.06,Z 178.024,A -85,B 0,C 180,E1 -11307.927,E2 -11307.927} C_VEL
LIN {X 0,Y 397.097,Z 178.022,A -85,B 0,C 180,E1 -11311.454,E2 -11311.454} C_VEL
LIN {X 0,Y 397.133,Z 178.015,A -85,B 0,C 180,E1 -11314.487,E2 -11314.487} C_VEL
LIN {X 0,Y 397.147,Z 178.012,A -85,B 0,C 180,E1 -11318.184,E2 -11318.184} C_VEL
LIN {X 0,Y 397.151,Z 178.013,A -85,B 0,C 180,E1 -11321.426,E2 -11321.426} C_VEL
LIN {X 0,Y 397.16,Z 178.015,A -85,B 0,C 180,E1 -11324.607,E2 -11324.607} C_VEL
LIN {X 0,Y 397.207,Z 178.005,A -85,B 0,C 180,E1 -11327.742,E2 -11327.742} C_VEL
LIN {X 0,Y 397.236,Z 178.003,A -85,B 0,C 180,E1 -11330.838,E2 -11330.838} C_VEL
LIN {X 0,Y 397.378,Z 177.985,A -85,B 0,C 180,E1 -11333.909,E2 -11333.909} C_VEL
LIN {X 0,Y 397.422,Z 177.981,A -85,B 0,C 180,E1 -11337.973,E2 -11337.973} C_VEL
LIN {X 0,Y 397.551,Z 177.966,A -85,B 0,C 180,E1 -11340,E2 -11340} C_VEL
LIN {X 0,Y 397.367,Z 177.984,A -85,B 0,C 180,E1 -11343.042,E2 -11343.042} C_VEL
LIN {X 0,Y 397.329,Z 177.99,A -85,B 0,C 180,E1 -11346.595,E2 -11346.595} C_VEL
LIN {X 0,Y 397.229,Z 178.002,A -85,B 0,C 180,E1 -11349.163,E2 -11349.163} C_VEL
LIN {X 0,Y 397.195,Z 178.008,A -85,B 0,C 180,E1 -11352.259,E2 -11352.259} C_VEL
LIN {X 0,Y 397.166,Z 178.013,A -85,B 0,C 180,E1 -11355.393,E2 -11355.393} C_VEL
LIN {X 0,Y 397.145,Z 178.012,A -85,B 0,C 180,E1 -11358.575,E2 -11358.575} C_VEL
LIN {X 0,Y 397.076,Z 178.024,A -85,B 0,C 180,E1 -11361.82,E2 -11361.82} C_VEL
LIN {X 0,Y 397.138,Z 178.017,A -85,B 0,C 180,E1 -11365.133,E2 -11365.133} C_VEL
LIN {X 0,Y 397.146,Z 178.014,A -85,B 0,C 180,E1 -11367.778,E2 -11367.778} C_VEL
LIN {X 0,Y 397.067,Z 178.025,A -85,B 0,C 180,E1 -11370.884,E2 -11370.884} C_VEL
LIN {X 0,Y 397.11,Z 178.018,A -85,B 0,C 180,E1 -11374.495,E2 -11374.495} C_VEL
LIN {X 0,Y 397.087,Z 178.02,A -85,B 0,C 180,E1 -11378.277,E2 -11378.277} C_VEL
LIN {X 0,Y 397.077,Z 178.027,A -85,B 0,C 180,E1 -11380.911,E2 -11380.911} C_VEL
LIN {X 0,Y 397.091,Z 178.019,A -85,B 0,C 180,E1 -11383.651,E2 -11383.651} C_VEL
LIN {X 0,Y 397.094,Z 178.024,A -85,B 0,C 180,E1 -11386.523,E2 -11386.523} C_VEL
LIN {X 0,Y 397.069,Z 178.026,A -85,B 0,C 180,E1 -11390.42,E2 -11390.42} C_VEL
LIN {X 0,Y 397.037,Z 178.137,A -85,B 0,C 180,E1 -11391.72,E2 -11391.72} C_VEL
LIN {X 0,Y 397.04,Z 181.407,A -85,B 0,C 180,E1 -11394.514,E2 -11394.514} C_VEL
LIN {X 0,Y 396.82,Z 185.47,A -85,B 0,C 180,E1 -11397.907,E2 -11397.907} C_VEL
LIN {X 0,Y 396.614,Z 189.843,A -85,B 0,C 180,E1 -11401.418,E2 -11401.418} C_VEL
LIN {X 0,Y 396.426,Z 194.294,A -85,B 0,C 180,E1 -11404.82,E2 -11404.82} C_VEL
LIN {X 0,Y 396.25,Z 198.708,A -85,B 0,C 180,E1 -11408.133,E2 -11408.133} C_VEL
LIN {X 0,Y 396.2,Z 200.778,A -85,B 0,C 180,E1 -11409.647,E2 -11409.647} C_VEL
LIN {X 0,Y 399.469,Z 213.818,A -85,B 0,C 180,E1 -11410.261,E2 -11410.261} C_VEL
LIN {X 0,Y 401.751,Z 225.333,A -85,B 0,C 180,E1 -11410.952,E2 -11410.952} C_VEL
LIN {X 0,Y 401.649,Z 233.134,A -85,B 0,C 180,E1 -11411.445,E2 -11411.445} C_VEL
LIN {X 0,Y 400.792,Z 245.321,A -85,B 0,C 180,E1 -11412.394,E2 -11412.394} C_VEL
LIN {X 0,Y 399.912,Z 255.62,A -85,B 0,C 180,E1 -11413.407,E2 -11413.407} C_VEL
LIN {X 0,Y 399.023,Z 266.012,A -85,B 0,C 180,E1 -11414.681,E2 -11414.681} C_VEL
LIN {X 0,Y 398.031,Z 275.844,A -85,B 0,C 180,E1 -11416.202,E2 -11416.202} C_VEL
LIN {X 0,Y 397.481,Z 283.826,A -85,B 0,C 180,E1 -11417.75,E2 -11417.75} C_VEL
LIN {X 0,Y 396.781,Z 290.16,A -85,B 0,C 180,E1 -11419.282,E2 -11419.282} C_VEL
LIN {X 0,Y 396.42,Z 295.182,A -85,B 0,C 180,E1 -11420.819,E2 -11420.819} C_VEL
LIN {X 0,Y 396.126,Z 299.074,A -85,B 0,C 180,E1 -11422.353,E2 -11422.353} C_VEL
LIN {X 0,Y 395.913,Z 301.941,A -85,B 0,C 180,E1 -11423.886,E2 -11423.886} C_VEL
LIN {X 0,Y 395.869,Z 303.293,A -85,B 0,C 180,E1 -11424.907,E2 -11424.907} C_VEL
LIN {X 0,Y 395.77,Z 304.833,A -85,B 0,C 180,E1 -11426.946,E2 -11426.946} C_VEL
LIN {X 0,Y 395.813,Z 305.011,A -85,B 0,C 180,E1 -11427.964,E2 -11427.964} C_VEL
LIN {X 0,Y 395.783,Z 304.151,A -85,B 0,C 180,E1 -11429.999,E2 -11429.999} C_VEL
LIN {X 0,Y 395.826,Z 303.149,A -85,B 0,C 180,E1 -11431.017,E2 -11431.017} C_VEL
LIN {X 0,Y 395.943,Z 301.738,A -85,B 0,C 180,E1 -11432.034,E2 -11432.034} C_VEL
LIN {X 0,Y 396.187,Z 298.811,A -85,B 0,C 180,E1 -11433.559,E2 -11433.559} C_VEL
LIN {X 0,Y 396.298,Z 294.86,A -85,B 0,C 180,E1 -11435.086,E2 -11435.086} C_VEL
LIN {X 0,Y 396.744,Z 289.761,A -85,B 0,C 180,E1 -11436.611,E2 -11436.611} C_VEL
LIN {X 0,Y 397.284,Z 282.125,A -85,B 0,C 180,E1 -11438.391,E2 -11438.391} C_VEL
LIN {X 0,Y 397.991,Z 273.884,A -85,B 0,C 180,E1 -11439.913,E2 -11439.913} C_VEL
LIN {X 0,Y 398.771,Z 265.404,A -85,B 0,C 180,E1 -11441.177,E2 -11441.177} C_VEL
LIN {X 0,Y 399.566,Z 254.944,A -85,B 0,C 180,E1 -11442.441,E2 -11442.441} C_VEL
LIN {X 0,Y 400.119,Z 245.999,A -85,B 0,C 180,E1 -11443.327,E2 -11443.327} C_VEL
LIN {X 0,Y 400.833,Z 236.705,A -85,B 0,C 180,E1 -11444.078,E2 -11444.078} C_VEL
LIN {X 0,Y 401.111,Z 231.243,A -85,B 0,C 180,E1 -11444.456,E2 -11444.456} C_VEL
LIN {X 0,Y 400.708,Z 226.843,A -85,B 0,C 180,E1 -11444.756,E2 -11444.756} C_VEL
LIN {X 0,Y 398.403,Z 221.036,A -85,B 0,C 180,E1 -11445.184,E2 -11445.184} C_VEL
LIN {X 0,Y 391.951,Z 209.713,A -85,B 0,C 180,E1 -11445.978,E2 -11445.978} C_VEL
LIN {X 0,Y 389.929,Z 204.322,A -85,B 0,C 180,E1 -11446.249,E2 -11446.249} C_VEL
LIN {X 0,Y 389.158,Z 200.91,A -85,B 0,C 180,E1 -11446.388,E2 -11446.388} C_VEL
LIN {X 0,Y 389.296,Z 195.85,A -85,B 0,C 180,E1 -11450.154,E2 -11450.154} C_VEL
LIN {X 0,Y 389.412,Z 191.59,A -85,B 0,C 180,E1 -11453.391,E2 -11453.391} C_VEL
LIN {X 0,Y 389.613,Z 187.256,A -85,B 0,C 180,E1 -11456.802,E2 -11456.802} C_VEL
LIN {X 0,Y 389.793,Z 182.963,A -85,B 0,C 180,E1 -11460.318,E2 -11460.318} C_VEL
LIN {X 0,Y 389.909,Z 180.082,A -85,B 0,C 180,E1 -11462.731,E2 -11462.731} C_VEL
LIN {X 0,Y 389.911,Z 178.921,A -85,B 0,C 180,E1 -11463.989,E2 -11463.989} C_VEL
LIN {X 0,Y 390.033,Z 178.898,A -85,B 0,C 180,E1 -11466.482,E2 -11466.482} C_VEL
LIN {X 0,Y 390.054,Z 178.9,A -85,B 0,C 180,E1 -11469.215,E2 -11469.215} C_VEL
LIN {X 0,Y 390.03,Z 178.899,A -85,B 0,C 180,E1 -11472.371,E2 -11472.371} C_VEL
LIN {X 0,Y 390.086,Z 178.891,A -85,B 0,C 180,E1 -11476.104,E2 -11476.104} C_VEL
LIN {X 0,Y 390.064,Z 178.899,A -85,B 0,C 180,E1 -11479.172,E2 -11479.172} C_VEL
LIN {X 0,Y 390.024,Z 178.901,A -85,B 0,C 180,E1 -11482.446,E2 -11482.446} C_VEL
LIN {X 0,Y 390.045,Z 178.897,A -85,B 0,C 180,E1 -11486.042,E2 -11486.042} C_VEL
LIN {X 0,Y 390.027,Z 178.899,A -85,B 0,C 180,E1 -11489.865,E2 -11489.865} C_VEL
LIN {X 0,Y 390.088,Z 178.892,A -85,B 0,C 180,E1 -11493.229,E2 -11493.229} C_VEL
LIN {X 0,Y 390.093,Z 178.894,A -85,B 0,C 180,E1 -11496.744,E2 -11496.744} C_VEL
LIN {X 0,Y 390.101,Z 178.892,A -85,B 0,C 180,E1 -11499.982,E2 -11499.982} C_VEL
LIN {X 0,Y 390.112,Z 178.889,A -85,B 0,C 180,E1 -11503.247,E2 -11503.247} C_VEL
LIN {X 0,Y 390.165,Z 178.885,A -85,B 0,C 180,E1 -11506.56,E2 -11506.56} C_VEL
LIN {X 0,Y 390.187,Z 178.881,A -85,B 0,C 180,E1 -11509.623,E2 -11509.623} C_VEL
LIN {X 0,Y 390.312,Z 178.863,A -85,B 0,C 180,E1 -11512.759,E2 -11512.759} C_VEL
LIN {X 0,Y 390.207,Z 178.876,A -85,B 0,C 180,E1 -11514.833,E2 -11514.833} C_VEL
LIN {X 0,Y 390.385,Z 178.859,A -85,B 0,C 180,E1 -11517.936,E2 -11517.936} C_VEL
LIN {X 0,Y 390.513,Z 178.843,A -85,B 0,C 180,E1 -11520,E2 -11520} C_VEL
LIN {X 0,Y 390.318,Z 178.864,A -85,B 0,C 180,E1 -11523.096,E2 -11523.096} C_VEL
LIN {X 0,Y 390.311,Z 178.865,A -85,B 0,C 180,E1 -11526.202,E2 -11526.202} C_VEL
LIN {X 0,Y 390.286,Z 178.867,A -85,B 0,C 180,E1 -11528.283,E2 -11528.283} C_VEL
LIN {X 0,Y 390.132,Z 178.891,A -85,B 0,C 180,E1 -11531.429,E2 -11531.429} C_VEL
LIN {X 0,Y 390.115,Z 178.889,A -85,B 0,C 180,E1 -11534.608,E2 -11534.608} C_VEL
LIN {X 0,Y 390.1,Z 178.891,A -85,B 0,C 180,E1 -11537.834,E2 -11537.834} C_VEL
LIN {X 0,Y 390.076,Z 178.898,A -85,B 0,C 180,E1 -11541.121,E2 -11541.121} C_VEL
LIN {X 0,Y 390.056,Z 178.897,A -85,B 0,C 180,E1 -11544.482,E2 -11544.482} C_VEL
LIN {X 0,Y 390.091,Z 178.89,A -85,B 0,C 180,E1 -11547.932,E2 -11547.932} C_VEL
LIN {X 0,Y 390.001,Z 178.903,A -85,B 0,C 180,E1 -11551.506,E2 -11551.506} C_VEL
LIN {X 0,Y 390.062,Z 178.896,A -85,B 0,C 180,E1 -11555.209,E2 -11555.209} C_VEL
LIN {X 0,Y 390.074,Z 178.894,A -85,B 0,C 180,E1 -11559.094,E2 -11559.094} C_VEL
LIN {X 0,Y 390.101,Z 178.895,A -85,B 0,C 180,E1 -11562.389,E2 -11562.389} C_VEL
LIN {X 0,Y 390.111,Z 178.894,A -85,B 0,C 180,E1 -11566.105,E2 -11566.105} C_VEL
LIN {X 0,Y 390.111,Z 179.105,A -85,B 0,C 180,E1 -11568.855,E2 -11568.855} C_VEL
LIN {X 0,Y 390.995,Z 184.462,A -85,B 0,C 180,E1 -11572.268,E2 -11572.268} C_VEL
LIN {X 0,Y 391.272,Z 187.207,A -85,B 0,C 180,E1 -11573.929,E2 -11573.929} C_VEL
LIN {X 0,Y 391.007,Z 192.155,A -85,B 0,C 180,E1 -11576.759,E2 -11576.759} C_VEL
LIN {X 0,Y 390.612,Z 197.567,A -85,B 0,C 180,E1 -11579.753,E2 -11579.753} C_VEL
LIN {X 0,Y 390.028,Z 205.149,A -85,B 0,C 180,E1 -11583.806,E2 -11583.806} C_VEL
LIN {X 0,Y 389.612,Z 212.686,A -85,B 0,C 180,E1 -11587.743,E2 -11587.743} C_VEL
LIN {X 0,Y 389.193,Z 220.156,A -85,B 0,C 180,E1 -11591.581,E2 -11591.581} C_VEL
LIN {X 0,Y 389.267,Z 221.096,A -85,B 0,C 180,E1 -11591.652,E2 -11591.652} C_VEL
LIN {X 0,Y 391.681,Z 234.109,A -85,B 0,C 180,E1 -11592.196,E2 -11592.196} C_VEL
LIN {X 0,Y 393.493,Z 247.371,A -85,B 0,C 180,E1 -11592.947,E2 -11592.947} C_VEL
LIN {X 0,Y 393.842,Z 253.003,A -85,B 0,C 180,E1 -11593.322,E2 -11593.322} C_VEL
LIN {X 0,Y 392.988,Z 264.406,A -85,B 0,C 180,E1 -11594.176,E2 -11594.176} C_VEL
LIN {X 0,Y 392.083,Z 275.15,A -85,B 0,C 180,E1 -11595.203,E2 -11595.203} C_VEL
LIN {X 0,Y 391.236,Z 285.926,A -85,B 0,C 180,E1 -11596.497,E2 -11596.497} C_VEL
LIN {X 0,Y 390.534,Z 294.679,A -85,B 0,C 180,E1 -11597.794,E2 -11597.794} C_VEL
LIN {X 0,Y 389.786,Z 303.179,A -85,B 0,C 180,E1 -11599.351,E2 -11599.351} C_VEL
LIN {X 0,Y 389.328,Z 310.008,A -85,B 0,C 180,E1 -11600.913,E2 -11600.913} C_VEL
LIN {X 0,Y 388.932,Z 316.281,A -85,B 0,C 180,E1 -11602.734,E2 -11602.734} C_VEL
LIN {X 0,Y 388.746,Z 320.179,A -85,B 0,C 180,E1 -11604.218,E2 -11604.218} C_VEL
LIN {X 0,Y 388.699,Z 323.392,A -85,B 0,C 180,E1 -11605.854,E2 -11605.854} C_VEL
LIN {X 0,Y 388.635,Z 324.879,A -85,B 0,C 180,E1 -11606.891,E2 -11606.891} C_VEL
LIN {X 0,Y 388.661,Z 325.924,A -85,B 0,C 180,E1 -11607.928,E2 -11607.928} C_VEL
LIN {X 0,Y 388.703,Z 326.581,A -85,B 0,C 180,E1 -11608.965,E2 -11608.965} C_VEL
LIN {X 0,Y 388.708,Z 326.851,A -85,B 0,C 180,E1 -11610.001,E2 -11610.001} C_VEL
LIN {X 0,Y 388.703,Z 326.72,A -85,B 0,C 180,E1 -11611.037,E2 -11611.037} C_VEL
LIN {X 0,Y 388.66,Z 326.158,A -85,B 0,C 180,E1 -11612.073,E2 -11612.073} C_VEL
LIN {X 0,Y 388.699,Z 323.867,A -85,B 0,C 180,E1 -11614.148,E2 -11614.148} C_VEL
LIN {X 0,Y 388.727,Z 320.928,A -85,B 0,C 180,E1 -11615.754,E2 -11615.754} C_VEL
LIN {X 0,Y 388.939,Z 317.164,A -85,B 0,C 180,E1 -11617.267,E2 -11617.267} C_VEL
LIN {X 0,Y 389.267,Z 312.179,A -85,B 0,C 180,E1 -11618.828,E2 -11618.828} C_VEL
LIN {X 0,Y 389.796,Z 305.923,A -85,B 0,C 180,E1 -11620.387,E2 -11620.387} C_VEL
LIN {X 0,Y 390.489,Z 298.105,A -85,B 0,C 180,E1 -11621.945,E2 -11621.945} C_VEL
LIN {X 0,Y 391.433,Z 288.352,A -85,B 0,C 180,E1 -11623.498,E2 -11623.498} C_VEL
LIN {X 0,Y 392.286,Z 278.481,A -85,B 0,C 180,E1 -11624.764,E2 -11624.764} C_VEL
LIN {X 0,Y 393.186,Z 268.242,A -85,B 0,C 180,E1 -11625.818,E2 -11625.818} C_VEL
LIN {X 0,Y 394.288,Z 255.879,A -85,B 0,C 180,E1 -11626.815,E2 -11626.815} C_VEL
LIN {X 0,Y 394.347,Z 250.582,A -85,B 0,C 180,E1 -11627.181,E2 -11627.181} C_VEL
LIN {X 0,Y 392.768,Z 238.2,A -85,B 0,C 180,E1 -11627.957,E2 -11627.957} C_VEL
LIN {X 0,Y 390.294,Z 225.194,A -85,B 0,C 180,E1 -11628.586,E2 -11628.586} C_VEL
LIN {X 0,Y 389.258,Z 220.159,A -85,B 0,C 180,E1 -11628.781,E2 -11628.781} C_VEL
LIN {X 0,Y 389.673,Z 213.425,A -85,B 0,C 180,E1 -11632.255,E2 -11632.255} C_VEL
LIN {X 0,Y 390.047,Z 206.892,A -85,B 0,C 180,E1 -11635.721,E2 -11635.721} C_VEL
LIN {X 0,Y 390.538,Z 200.687,A -85,B 0,C 180,E1 -11639.069,E2 -11639.069} C_VEL
LIN {X 0,Y 391.059,Z 194.27,A -85,B 0,C 180,E1 -11642.624,E2 -11642.624} C_VEL
LIN {X 0,Y 391.406,Z 190.025,A -85,B 0,C 180,E1 -11645.068,E2 -11645.068} C_VEL
LIN {X 0,Y 391.192,Z 185.599,A -85,B 0,C 180,E1 -11647.769,E2 -11647.769} C_VEL
LIN {X 0,Y 390.419,Z 180.842,A -85,B 0,C 180,E1 -11650.883,E2 -11650.883} C_VEL
LIN {X 0,Y 390.107,Z 178.892,A -85,B 0,C 180,E1 -11652.301,E2 -11652.301} C_VEL
LIN {X 0,Y 390.05,Z 178.9,A -85,B 0,C 180,E1 -11655.355,E2 -11655.355} C_VEL
LIN {X 0,Y 390.017,Z 178.901,A -85,B 0,C 180,E1 -11658.185,E2 -11658.185} C_VEL
LIN {X 0,Y 390.068,Z 178.895,A -85,B 0,C 180,E1 -11660.905,E2 -11660.905} C_VEL
LIN {X 0,Y 390.069,Z 178.894,A -85,B 0,C 180,E1 -11664.791,E2 -11664.791} C_VEL
LIN {X 0,Y 390.005,Z 178.902,A -85,B 0,C 180,E1 -11668.494,E2 -11668.494} C_VEL
LIN {X 0,Y 390.1,Z 178.89,A -85,B 0,C 180,E1 -11672.069,E2 -11672.069} C_VEL
LIN {X 0,Y 390.064,Z 178.896,A -85,B 0,C 180,E1 -11675.518,E2 -11675.518} C_VEL
LIN {X 0,Y 390.085,Z 178.897,A -85,B 0,C 180,E1 -11678.88,E2 -11678.88} C_VEL
LIN {X 0,Y 390.129,Z 178.892,A -85,B 0,C 180,E1 -11682.691,E2 -11682.691} C_VEL
LIN {X 0,Y 390.173,Z 178.886,A -85,B 0,C 180,E1 -11686.561,E2 -11686.561} C_VEL
LIN {X 0,Y 390.158,Z 178.882,A -85,B 0,C 180,E1 -11689.623,E2 -11689.623} C_VEL
LIN {X 0,Y 390.31,Z 178.867,A -85,B 0,C 180,E1 -11692.759,E2 -11692.759} C_VEL
LIN {X 0,Y 390.214,Z 178.878,A -85,B 0,C 180,E1 -11694.834,E2 -11694.834} C_VEL
LIN {X 0,Y 390.392,Z 178.856,A -85,B 0,C 180,E1 -11697.937,E2 -11697.937} C_VEL
LIN {X 0,Y 390.521,Z 178.842,A -85,B 0,C 180,E1 -11700,E2 -11700} C_VEL
LIN {X 0,Y 390.327,Z 178.861,A -85,B 0,C 180,E1 -11703.097,E2 -11703.097} C_VEL
LIN {X 0,Y 390.286,Z 178.868,A -85,B 0,C 180,E1 -11706.588,E2 -11706.588} C_VEL
LIN {X 0,Y 390.181,Z 178.881,A -85,B 0,C 180,E1 -11709.33,E2 -11709.33} C_VEL
LIN {X 0,Y 390.173,Z 178.884,A -85,B 0,C 180,E1 -11713.439,E2 -11713.439} C_VEL
LIN {X 0,Y 390.143,Z 178.887,A -85,B 0,C 180,E1 -11717.316,E2 -11717.316} C_VEL
LIN {X 0,Y 390.036,Z 178.9,A -85,B 0,C 180,E1 -11721.124,E2 -11721.124} C_VEL
LIN {X 0,Y 390.061,Z 178.895,A -85,B 0,C 180,E1 -11724.482,E2 -11724.482} C_VEL
LIN {X 0,Y 390.101,Z 178.89,A -85,B 0,C 180,E1 -11727.932,E2 -11727.932} C_VEL
LIN {X 0,Y 390.011,Z 178.904,A -85,B 0,C 180,E1 -11731.506,E2 -11731.506} C_VEL
LIN {X 0,Y 390.071,Z 178.898,A -85,B 0,C 180,E1 -11735.209,E2 -11735.209} C_VEL
LIN {X 0,Y 390.055,Z 178.899,A -85,B 0,C 180,E1 -11739.22,E2 -11739.22} C_VEL
LIN {X 0,Y 390.031,Z 178.9,A -85,B 0,C 180,E1 -11742.376,E2 -11742.376} C_VEL
LIN {X 0,Y 390.035,Z 178.899,A -85,B 0,C 180,E1 -11745.356,E2 -11745.356} C_VEL
LIN {X 0,Y 390.018,Z 178.902,A -85,B 0,C 180,E1 -11748.188,E2 -11748.188} C_VEL
LIN {X 0,Y 390.031,Z 178.904,A -85,B 0,C 180,E1 -11750.903,E2 -11750.903} C_VEL
LIN {X 0,Y 390.018,Z 179.968,A -85,B 0,C 180,E1 -11752.455,E2 -11752.455} C_VEL
LIN {X 0,Y 389.999,Z 182.67,A -85,B 0,C 180,E1 -11754.786,E2 -11754.786} C_VEL
LIN {X 0,Y 389.745,Z 187.055,A -85,B 0,C 180,E1 -11758.472,E2 -11758.472} C_VEL
LIN {X 0,Y 389.605,Z 189.975,A -85,B 0,C 180,E1 -11760.855,E2 -11760.855} C_VEL
LIN {X 0,Y 389.413,Z 194.606,A -85,B 0,C 180,E1 -11764.474,E2 -11764.474} C_VEL
LIN {X 0,Y 389.211,Z 198.88,A -85,B 0,C 180,E1 -11767.717,E2 -11767.717} C_VEL
LIN {X 0,Y 389.139,Z 200.971,A -85,B 0,C 180,E1 -11769.286,E2 -11769.286} C_VEL
LIN {X 0,Y 392.535,Z 214.206,A -85,B 0,C 180,E1 -11769.929,E2 -11769.929} C_VEL
LIN {X 0,Y 395.024,Z 226.95,A -85,B 0,C 180,E1 -11770.722,E2 -11770.722} C_VEL
LIN {X 0,Y 394.626,Z 237.469,A -85,B 0,C 180,E1 -11771.438,E2 -11771.438} C_VEL
LIN {X 0,Y 393.74,Z 248.13,A -85,B 0,C 180,E1 -11772.336,E2 -11772.336} C_VEL
LIN {X 0,Y 392.741,Z 258.995,A -85,B 0,C 180,E1 -11773.497,E2 -11773.497} C_VEL
LIN {X 0,Y 391.943,Z 267.846,A -85,B 0,C 180,E1 -11774.664,E2 -11774.664} C_VEL
LIN {X 0,Y 391.06,Z 276.439,A -85,B 0,C 180,E1 -11776.044,E2 -11776.044} C_VEL
LIN {X 0,Y 390.486,Z 283.923,A -85,B 0,C 180,E1 -11777.527,E2 -11777.527} C_VEL
LIN {X 0,Y 389.759,Z 290.283,A -85,B 0,C 180,E1 -11779.086,E2 -11779.086} C_VEL
LIN {X 0,Y 389.37,Z 295.321,A -85,B 0,C 180,E1 -11780.651,E2 -11780.651} C_VEL
LIN {X 0,Y 389.064,Z 299.228,A -85,B 0,C 180,E1 -11782.214,E2 -11782.214} C_VEL
LIN {X 0,Y 388.857,Z 302.108,A -85,B 0,C 180,E1 -11783.774,E2 -11783.774} C_VEL
LIN {X 0,Y 388.788,Z 303.467,A -85,B 0,C 180,E1 -11784.814,E2 -11784.814} C_VEL
LIN {X 0,Y 388.674,Z 305.021,A -85,B 0,C 180,E1 -11786.89,E2 -11786.89} C_VEL
LIN {X 0,Y 388.713,Z 305.211,A -85,B 0,C 180,E1 -11787.927,E2 -11787.927} C_VEL
LIN {X 0,Y 388.728,Z 304.977,A -85,B 0,C 180,E1 -11788.963,E2 -11788.963} C_VEL
LIN {X 0,Y 388.757,Z 303.369,A -85,B 0,C 180,E1 -11791.035,E2 -11791.035} C_VEL
LIN {X 0,Y 388.88,Z 301.97,A -85,B 0,C 180,E1 -11792.071,E2 -11792.071} C_VEL
LIN {X 0,Y 389.126,Z 299.054,A -85,B 0,C 180,E1 -11793.623,E2 -11793.623} C_VEL
LIN {X 0,Y 389.241,Z 295.118,A -85,B 0,C 180,E1 -11795.179,E2 -11795.179} C_VEL
LIN {X 0,Y 389.696,Z 290.039,A -85,B 0,C 180,E1 -11796.731,E2 -11796.731} C_VEL
LIN {X 0,Y 390.183,Z 283.646,A -85,B 0,C 180,E1 -11798.284,E2 -11798.284} C_VEL
LIN {X 0,Y 390.846,Z 275.682,A -85,B 0,C 180,E1 -11799.834,E2 -11799.834} C_VEL
LIN {X 0,Y 391.645,Z 267.553,A -85,B 0,C 180,E1 -11801.121,E2 -11801.121} C_VEL
LIN {X 0,Y 392.463,Z 257.643,A -85,B 0,C 180,E1 -11802.407,E2 -11802.407} C_VEL
LIN {X 0,Y 393.232,Z 246.43,A -85,B 0,C 180,E1 -11803.565,E2 -11803.565} C_VEL
LIN {X 0,Y 393.98,Z 237.191,A -85,B 0,C 180,E1 -11804.328,E2 -11804.328} C_VEL
LIN {X 0,Y 394.465,Z 226.562,A -85,B 0,C 180,E1 -11805.04,E2 -11805.04} C_VEL
LIN {X 0,Y 391.969,Z 213.25,A -85,B 0,C 180,E1 -11805.834,E2 -11805.834} C_VEL
LIN {X 0,Y 389.929,Z 204.322,A -85,B 0,C 180,E1 -11806.249,E2 -11806.249} C_VEL
LIN {X 0,Y 389.001,Z 202.029,A -85,B 0,C 180,E1 -11806.473,E2 -11806.473} C_VEL
LIN {X 0,Y 387.552,Z 200.319,A -85,B 0,C 180,E1 -11806.939,E2 -11806.939} C_VEL
LIN {X 0,Y 383.929,Z 198.562,A -85,B 0,C 180,E1 -11808.633,E2 -11808.633} C_VEL
LIN {X 0,Y 382.439,Z 196.893,A -85,B 0,C 180,E1 -11809.938,E2 -11809.938} C_VEL
LIN {X 0,Y 382.229,Z 195.999,A -85,B 0,C 180,E1 -11810.599,E2 -11810.599} C_VEL
LIN {X 0,Y 382.368,Z 191.781,A -85,B 0,C 180,E1 -11813.849,E2 -11813.849} C_VEL
LIN {X 0,Y 382.571,Z 187.441,A -85,B 0,C 180,E1 -11817.336,E2 -11817.336} C_VEL
LIN {X 0,Y 382.793,Z 183.119,A -85,B 0,C 180,E1 -11820.932,E2 -11820.932} C_VEL
LIN {X 0,Y 382.839,Z 180.248,A -85,B 0,C 180,E1 -11823.413,E2 -11823.413} C_VEL
LIN {X 0,Y 382.899,Z 179.79,A -85,B 0,C 180,E1 -11824.677,E2 -11824.677} C_VEL
LIN {X 0,Y 382.979,Z 179.781,A -85,B 0,C 180,E1 -11827.266,E2 -11827.266} C_VEL
LIN {X 0,Y 382.995,Z 179.776,A -85,B 0,C 180,E1 -11829.956,E2 -11829.956} C_VEL
LIN {X 0,Y 382.992,Z 179.777,A -85,B 0,C 180,E1 -11832.776,E2 -11832.776} C_VEL
LIN {X 0,Y 383.022,Z 179.772,A -85,B 0,C 180,E1 -11835.792,E2 -11835.792} C_VEL
LIN {X 0,Y 383.026,Z 179.773,A -85,B 0,C 180,E1 -11838.784,E2 -11838.784} C_VEL
LIN {X 0,Y 382.981,Z 179.777,A -85,B 0,C 180,E1 -11842.093,E2 -11842.093} C_VEL
LIN {X 0,Y 382.996,Z 179.777,A -85,B 0,C 180,E1 -11845.329,E2 -11845.329} C_VEL
LIN {X 0,Y 382.962,Z 179.782,A -85,B 0,C 180,E1 -11849.079,E2 -11849.079} C_VEL
LIN {X 0,Y 383.032,Z 179.776,A -85,B 0,C 180,E1 -11852.696,E2 -11852.696} C_VEL
LIN {X 0,Y 383.02,Z 179.774,A -85,B 0,C 180,E1 -11856.191,E2 -11856.191} C_VEL
LIN {X 0,Y 383.053,Z 179.768,A -85,B 0,C 180,E1 -11859.598,E2 -11859.598} C_VEL
LIN {X 0,Y 383.077,Z 179.766,A -85,B 0,C 180,E1 -11862.93,E2 -11862.93} C_VEL
LIN {X 0,Y 383.096,Z 179.766,A -85,B 0,C 180,E1 -11866.462,E2 -11866.462} C_VEL
LIN {X 0,Y 383.141,Z 179.757,A -85,B 0,C 180,E1 -11869.43,E2 -11869.43} C_VEL
LIN {X 0,Y 383.263,Z 179.742,A -85,B 0,C 180,E1 -11872.625,E2 -11872.625} C_VEL
LIN {X 0,Y 383.179,Z 179.752,A -85,B 0,C 180,E1 -11874.738,E2 -11874.738} C_VEL
LIN {X 0,Y 383.353,Z 179.735,A -85,B 0,C 180,E1 -11877.898,E2 -11877.898} C_VEL
LIN {X 0,Y 383.483,Z 179.718,A -85,B 0,C 180,E1 -11880,E2 -11880} C_VEL
LIN {X 0,Y 383.253,Z 179.745,A -85,B 0,C 180,E1 -11883.153,E2 -11883.153} C_VEL
LIN {X 0,Y 383.266,Z 179.741,A -85,B 0,C 180,E1 -11886.316,E2 -11886.316} C_VEL
LIN {X 0,Y 383.232,Z 179.745,A -85,B 0,C 180,E1 -11888.436,E2 -11888.436} C_VEL
LIN {X 0,Y 383.08,Z 179.768,A -85,B 0,C 180,E1 -11891.642,E2 -11891.642} C_VEL
LIN {X 0,Y 383.081,Z 179.767,A -85,B 0,C 180,E1 -11894.883,E2 -11894.883} C_VEL
LIN {X 0,Y 383.064,Z 179.767,A -85,B 0,C 180,E1 -11898.173,E2 -11898.173} C_VEL
LIN {X 0,Y 383.041,Z 179.771,A -85,B 0,C 180,E1 -11901.528,E2 -11901.528} C_VEL
LIN {X 0,Y 383.027,Z 179.776,A -85,B 0,C 180,E1 -11904.962,E2 -11904.962} C_VEL
LIN {X 0,Y 383.016,Z 179.774,A -85,B 0,C 180,E1 -11908.495,E2 -11908.495} C_VEL
LIN {X 0,Y 382.985,Z 179.777,A -85,B 0,C 180,E1 -11912.152,E2 -11912.152} C_VEL
LIN {X 0,Y 382.995,Z 179.78,A -85,B 0,C 180,E1 -11914.67,E2 -11914.67} C_VEL
LIN {X 0,Y 382.981,Z 179.778,A -85,B 0,C 180,E1 -11917.907,E2 -11917.907} C_VEL
LIN {X 0,Y 383.027,Z 179.771,A -85,B 0,C 180,E1 -11921.342,E2 -11921.342} C_VEL
LIN {X 0,Y 383.051,Z 179.774,A -85,B 0,C 180,E1 -11924.317,E2 -11924.317} C_VEL
LIN {X 0,Y 383.046,Z 179.776,A -85,B 0,C 180,E1 -11927.962,E2 -11927.962} C_VEL
LIN {X 0,Y 383.048,Z 179.83,A -85,B 0,C 180,E1 -11928.49,E2 -11928.49} C_VEL
LIN {X 0,Y 383.912,Z 185.078,A -85,B 0,C 180,E1 -11931.922,E2 -11931.922} C_VEL
LIN {X 0,Y 384.242,Z 188.746,A -85,B 0,C 180,E1 -11934.18,E2 -11934.18} C_VEL
LIN {X 0,Y 384.002,Z 193.065,A -85,B 0,C 180,E1 -11936.701,E2 -11936.701} C_VEL
LIN {X 0,Y 383.61,Z 197.912,A -85,B 0,C 180,E1 -11939.437,E2 -11939.437} C_VEL
LIN {X 0,Y 383.103,Z 203.874,A -85,B 0,C 180,E1 -11942.705,E2 -11942.705} C_VEL
LIN {X 0,Y 382.664,Z 210.327,A -85,B 0,C 180,E1 -11946.171,E2 -11946.171} C_VEL
LIN {X 0,Y 382.32,Z 216.746,A -85,B 0,C 180,E1 -11949.56,E2 -11949.56} C_VEL
LIN {X 0,Y 382.141,Z 220.192,A -85,B 0,C 180,E1 -11951.298,E2 -11951.298} C_VEL
LIN {X 0,Y 384.583,Z 233.491,A -85,B 0,C 180,E1 -11951.854,E2 -11951.854} C_VEL
LIN {X 0,Y 386.311,Z 246.121,A -85,B 0,C 180,E1 -11952.574,E2 -11952.574} C_VEL
LIN {X 0,Y 386.997,Z 252.691,A -85,B 0,C 180,E1 -11953.026,E2 -11953.026} C_VEL
LIN {X 0,Y 386.129,Z 264.035,A -85,B 0,C 180,E1 -11953.887,E2 -11953.887} C_VEL
LIN {X 0,Y 385.205,Z 274.82,A -85,B 0,C 180,E1 -11954.932,E2 -11954.932} C_VEL
LIN {X 0,Y 384.308,Z 285.618,A -85,B 0,C 180,E1 -11956.249,E2 -11956.249} C_VEL
LIN {X 0,Y 383.566,Z 294.39,A -85,B 0,C 180,E1 -11957.569,E2 -11957.569} C_VEL
LIN {X 0,Y 382.751,Z 302.911,A -85,B 0,C 180,E1 -11959.153,E2 -11959.153} C_VEL
LIN {X 0,Y 382.261,Z 309.752,A -85,B 0,C 180,E1 -11960.744,E2 -11960.744} C_VEL
LIN {X 0,Y 381.861,Z 316.038,A -85,B 0,C 180,E1 -11962.599,E2 -11962.599} C_VEL
LIN {X 0,Y 381.693,Z 319.388,A -85,B 0,C 180,E1 -11963.873,E2 -11963.873} C_VEL
LIN {X 0,Y 381.625,Z 323.17,A -85,B 0,C 180,E1 -11965.777,E2 -11965.777} C_VEL
LIN {X 0,Y 381.547,Z 324.665,A -85,B 0,C 180,E1 -11966.833,E2 -11966.833} C_VEL
LIN {X 0,Y 381.617,Z 326.377,A -85,B 0,C 180,E1 -11968.946,E2 -11968.946} C_VEL
LIN {X 0,Y 381.639,Z 326.651,A -85,B 0,C 180,E1 -11970.001,E2 -11970.001} C_VEL
LIN {X 0,Y 381.602,Z 326.527,A -85,B 0,C 180,E1 -11971.056,E2 -11971.056} C_VEL
LIN {X 0,Y 381.546,Z 325.026,A -85,B 0,C 180,E1 -11973.168,E2 -11973.168} C_VEL
LIN {X 0,Y 381.624,Z 323.689,A -85,B 0,C 180,E1 -11974.225,E2 -11974.225} C_VEL
LIN {X 0,Y 381.67,Z 320.274,A -85,B 0,C 180,E1 -11976.094,E2 -11976.094} C_VEL
LIN {X 0,Y 381.979,Z 315.477,A -85,B 0,C 180,E1 -11977.932,E2 -11977.932} C_VEL
LIN {X 0,Y 382.479,Z 309.08,A -85,B 0,C 180,E1 -11979.786,E2 -11979.786} C_VEL
LIN {X 0,Y 383.067,Z 302.111,A -85,B 0,C 180,E1 -11981.375,E2 -11981.375} C_VEL
LIN {X 0,Y 384.03,Z 293.388,A -85,B 0,C 180,E1 -11982.955,E2 -11982.955} C_VEL
LIN {X 0,Y 384.811,Z 284.367,A -85,B 0,C 180,E1 -11984.287,E2 -11984.287} C_VEL
LIN {X 0,Y 385.876,Z 273.454,A -85,B 0,C 180,E1 -11985.583,E2 -11985.583} C_VEL
LIN {X 0,Y 386.902,Z 262.309,A -85,B 0,C 180,E1 -11986.624,E2 -11986.624} C_VEL
LIN {X 0,Y 387.601,Z 252.636,A -85,B 0,C 180,E1 -11987.351,E2 -11987.351} C_VEL
LIN {X 0,Y 386.134,Z 240.258,A -85,B 0,C 180,E1 -11988.174,E2 -11988.174} C_VEL
LIN {X 0,Y 383.809,Z 227.462,A -85,B 0,C 180,E1 -11988.849,E2 -11988.849} C_VEL
LIN {X 0,Y 382.219,Z 219.933,A -85,B 0,C 180,E1 -11989.166,E2 -11989.166} C_VEL
LIN {X 0,Y 382.645,Z 213.286,A -85,B 0,C 180,E1 -11992.687,E2 -11992.687} C_VEL
LIN {X 0,Y 383.028,Z 206.948,A -85,B 0,C 180,E1 -11996.126,E2 -11996.126} C_VEL
LIN {X 0,Y 383.592,Z 200.566,A -85,B 0,C 180,E1 -11999.647,E2 -11999.647} C_VEL
LIN {X 0,Y 384.032,Z 195.248,A -85,B 0,C 180,E1 -12002.667,E2 -12002.667} C_VEL
LIN {X 0,Y 384.359,Z 191.871,A -85,B 0,C 180,E1 -12004.631,E2 -12004.631} C_VEL
LIN {X 0,Y 384.299,Z 187.819,A -85,B 0,C 180,E1 -12007.119,E2 -12007.119} C_VEL
LIN {X 0,Y 383.516,Z 182.59,A -85,B 0,C 180,E1 -12010.567,E2 -12010.567} C_VEL
LIN {X 0,Y 383.075,Z 179.766,A -85,B 0,C 180,E1 -12012.569,E2 -12012.569} C_VEL
LIN {X 0,Y 382.996,Z 179.78,A -85,B 0,C 180,E1 -12015.789,E2 -12015.789} C_VEL
LIN {X 0,Y 382.974,Z 179.777,A -85,B 0,C 180,E1 -12018.795,E2 -12018.795} C_VEL
LIN {X 0,Y 382.982,Z 179.777,A -85,B 0,C 180,E1 -12022.095,E2 -12022.095} C_VEL
LIN {X 0,Y 383.002,Z 179.78,A -85,B 0,C 180,E1 -12025.331,E2 -12025.331} C_VEL
LIN {X 0,Y 382.965,Z 179.783,A -85,B 0,C 180,E1 -12029.08,E2 -12029.08} C_VEL
LIN {X 0,Y 383.038,Z 179.771,A -85,B 0,C 180,E1 -12032.697,E2 -12032.697} C_VEL
LIN {X 0,Y 383.027,Z 179.771,A -85,B 0,C 180,E1 -12036.192,E2 -12036.192} C_VEL
LIN {X 0,Y 383.061,Z 179.767,A -85,B 0,C 180,E1 -12039.599,E2 -12039.599} C_VEL
LIN {X 0,Y 383.085,Z 179.768,A -85,B 0,C 180,E1 -12042.931,E2 -12042.931} C_VEL
LIN {X 0,Y 383.104,Z 179.765,A -85,B 0,C 180,E1 -12046.463,E2 -12046.463} C_VEL
LIN {X 0,Y 383.12,Z 179.759,A -85,B 0,C 180,E1 -12049.43,E2 -12049.43} C_VEL
LIN {X 0,Y 383.256,Z 179.747,A -85,B 0,C 180,E1 -12052.625,E2 -12052.625} C_VEL
LIN {X 0,Y 383.187,Z 179.753,A -85,B 0,C 180,E1 -12054.739,E2 -12054.739} C_VEL
LIN {X 0,Y 383.36,Z 179.732,A -85,B 0,C 180,E1 -12057.899,E2 -12057.899} C_VEL
LIN {X 0,Y 383.49,Z 179.717,A -85,B 0,C 180,E1 -12060,E2 -12060} C_VEL
LIN {X 0,Y 383.262,Z 179.741,A -85,B 0,C 180,E1 -12063.154,E2 -12063.154} C_VEL
LIN {X 0,Y 383.246,Z 179.744,A -85,B 0,C 180,E1 -12066.578,E2 -12066.578} C_VEL
LIN {X 0,Y 383.128,Z 179.76,A -85,B 0,C 180,E1 -12069.503,E2 -12069.503} C_VEL
LIN {X 0,Y 383.104,Z 179.765,A -85,B 0,C 180,E1 -12073.537,E2 -12073.537} C_VEL
LIN {X 0,Y 383.087,Z 179.767,A -85,B 0,C 180,E1 -12077.462,E2 -12077.462} C_VEL
LIN {X 0,Y 383.009,Z 179.773,A -85,B 0,C 180,E1 -12080.648,E2 -12080.648} C_VEL
LIN {X 0,Y 383.015,Z 179.775,A -85,B 0,C 180,E1 -12083.809,E2 -12083.809} C_VEL
LIN {X 0,Y 383.062,Z 179.766,A -85,B 0,C 180,E1 -12086.125,E2 -12086.125} C_VEL
LIN {X 0,Y 383.026,Z 179.771,A -85,B 0,C 180,E1 -12088.494,E2 -12088.494} C_VEL
LIN {X 0,Y 382.995,Z 179.774,A -85,B 0,C 180,E1 -12092.152,E2 -12092.152} C_VEL
LIN {X 0,Y 383.004,Z 179.776,A -85,B 0,C 180,E1 -12094.67,E2 -12094.67} C_VEL
LIN {X 0,Y 382.985,Z 179.776,A -85,B 0,C 180,E1 -12097.905,E2 -12097.905} C_VEL
LIN {X 0,Y 382.972,Z 179.779,A -85,B 0,C 180,E1 -12101.35,E2 -12101.35} C_VEL
LIN {X 0,Y 382.986,Z 179.777,A -85,B 0,C 180,E1 -12104.305,E2 -12104.305} C_VEL
LIN {X 0,Y 383.003,Z 179.775,A -85,B 0,C 180,E1 -12107.242,E2 -12107.242} C_VEL
LIN {X 0,Y 382.968,Z 179.783,A -85,B 0,C 180,E1 -12110.423,E2 -12110.423} C_VEL
LIN {X 0,Y 382.939,Z 179.809,A -85,B 0,C 180,E1 -12111.394,E2 -12111.394} C_VEL
LIN {X 0,Y 382.982,Z 182.749,A -85,B 0,C 180,E1 -12114.042,E2 -12114.042} C_VEL
LIN {X 0,Y 382.807,Z 185.727,A -85,B 0,C 180,E1 -12116.582,E2 -12116.582} C_VEL
LIN {X 0,Y 382.583,Z 190.107,A -85,B 0,C 180,E1 -12120.267,E2 -12120.267} C_VEL
LIN {X 0,Y 382.372,Z 195.111,A -85,B 0,C 180,E1 -12124.241,E2 -12124.241} C_VEL
LIN {X 0,Y 382.203,Z 199.03,A -85,B 0,C 180,E1 -12127.286,E2 -12127.286} C_VEL
LIN {X 0,Y 382.097,Z 201.158,A -85,B 0,C 180,E1 -12128.902,E2 -12128.902} C_VEL
LIN {X 0,Y 385.719,Z 215.32,A -85,B 0,C 180,E1 -12129.623,E2 -12129.623} C_VEL
LIN {X 0,Y 388.251,Z 228.113,A -85,B 0,C 180,E1 -12130.453,E2 -12130.453} C_VEL
LIN {X 0,Y 387.749,Z 239.096,A -85,B 0,C 180,E1 -12131.234,E2 -12131.234} C_VEL
LIN {X 0,Y 386.738,Z 250.717,A -85,B 0,C 180,E1 -12132.279,E2 -12132.279} C_VEL
LIN {X 0,Y 385.763,Z 261.156,A -85,B 0,C 180,E1 -12133.462,E2 -12133.462} C_VEL
LIN {X 0,Y 384.9,Z 269.678,A -85,B 0,C 180,E1 -12134.648,E2 -12134.648} C_VEL
LIN {X 0,Y 384.103,Z 276.999,A -85,B 0,C 180,E1 -12135.874,E2 -12135.874} C_VEL
LIN {X 0,Y 383.518,Z 284.021,A -85,B 0,C 180,E1 -12137.297,E2 -12137.297} C_VEL
LIN {X 0,Y 382.756,Z 290.406,A -85,B 0,C 180,E1 -12138.884,E2 -12138.884} C_VEL
LIN {X 0,Y 382.334,Z 295.461,A -85,B 0,C 180,E1 -12140.477,E2 -12140.477} C_VEL
LIN {X 0,Y 382.025,Z 299.383,A -85,B 0,C 180,E1 -12142.069,E2 -12142.069} C_VEL
LIN {X 0,Y 381.768,Z 302.435,A -85,B 0,C 180,E1 -12143.774,E2 -12143.774} C_VEL
LIN {X 0,Y 381.643,Z 304.617,A -85,B 0,C 180,E1 -12145.775,E2 -12145.775} C_VEL
LIN {X 0,Y 381.612,Z 305.41,A -85,B 0,C 180,E1 -12147.889,E2 -12147.889} C_VEL
LIN {X 0,Y 381.642,Z 305.185,A -85,B 0,C 180,E1 -12148.944,E2 -12148.944} C_VEL
LIN {X 0,Y 381.69,Z 303.589,A -85,B 0,C 180,E1 -12151.054,E2 -12151.054} C_VEL
LIN {X 0,Y 381.799,Z 302.202,A -85,B 0,C 180,E1 -12152.109,E2 -12152.109} C_VEL
LIN {X 0,Y 382.046,Z 299.298,A -85,B 0,C 180,E1 -12153.691,E2 -12153.691} C_VEL
LIN {X 0,Y 382.189,Z 295.375,A -85,B 0,C 180,E1 -12155.274,E2 -12155.274} C_VEL
LIN {X 0,Y 382.729,Z 289.325,A -85,B 0,C 180,E1 -12157.119,E2 -12157.119} C_VEL
LIN {X 0,Y 383.242,Z 282.723,A -85,B 0,C 180,E1 -12158.7,E2 -12158.7} C_VEL
LIN {X 0,Y 384.047,Z 274.523,A -85,B 0,C 180,E1 -12160.276,E2 -12160.276} C_VEL
LIN {X 0,Y 384.904,Z 266.111,A -85,B 0,C 180,E1 -12161.585,E2 -12161.585} C_VEL
LIN {X 0,Y 385.762,Z 255.721,A -85,B 0,C 180,E1 -12162.894,E2 -12162.894} C_VEL
LIN {X 0,Y 386.355,Z 246.859,A -85,B 0,C 180,E1 -12163.811,E2 -12163.811} C_VEL
LIN {X 0,Y 387.136,Z 237.674,A -85,B 0,C 180,E1 -12164.587,E2 -12164.587} C_VEL
LIN {X 0,Y 387.579,Z 227.406,A -85,B 0,C 180,E1 -12165.297,E2 -12165.297} C_VEL
LIN {X 0,Y 385.114,Z 214.212,A -85,B 0,C 180,E1 -12166.111,E2 -12166.111} C_VEL
LIN {X 0,Y 382.107,Z 201.102,A -85,B 0,C 180,E1 -12166.733,E2 -12166.733} C_VEL
LIN {X 0,Y 382.229,Z 195.999,A -85,B 0,C 180,E1 -12170.599,E2 -12170.599} C_VEL
LIN {X 0,Y 381.574,Z 194.939,A -85,B 0,C 180,E1 -12171.465,E2 -12171.465} C_VEL
LIN {X 0,Y 378.744,Z 193.422,A -85,B 0,C 180,E1 -12172.88,E2 -12172.88} C_VEL
LIN {X 0,Y 376.383,Z 192.241,A -85,B 0,C 180,E1 -12174.025,E2 -12174.025} C_VEL
LIN {X 0,Y 375.425,Z 191.245,A -85,B 0,C 180,E1 -12174.907,E2 -12174.907} C_VEL
LIN {X 0,Y 375.376,Z 190.88,A -85,B 0,C 180,E1 -12175.205,E2 -12175.205} C_VEL
LIN {X 0,Y 375.583,Z 186.985,A -85,B 0,C 180,E1 -12178.42,E2 -12178.42} C_VEL
LIN {X 0,Y 375.782,Z 183.306,A -85,B 0,C 180,E1 -12181.575,E2 -12181.575} C_VEL
LIN {X 0,Y 375.809,Z 180.676,A -85,B 0,C 180,E1 -12184.123,E2 -12184.123} C_VEL
LIN {X 0,Y 375.934,Z 180.655,A -85,B 0,C 180,E1 -12186.739,E2 -12186.739} C_VEL
LIN {X 0,Y 375.975,Z 180.65,A -85,B 0,C 180,E1 -12189.967,E2 -12189.967} C_VEL
LIN {X 0,Y 375.923,Z 180.657,A -85,B 0,C 180,E1 -12193.762,E2 -12193.762} C_VEL
LIN {X 0,Y 375.973,Z 180.652,A -85,B 0,C 180,E1 -12196.799,E2 -12196.799} C_VEL
LIN {X 0,Y 375.98,Z 180.648,A -85,B 0,C 180,E1 -12200.025,E2 -12200.025} C_VEL
LIN {X 0,Y 375.943,Z 180.655,A -85,B 0,C 180,E1 -12203.493,E2 -12203.493} C_VEL
LIN {X 0,Y 375.938,Z 180.654,A -85,B 0,C 180,E1 -12205.886,E2 -12205.886} C_VEL
LIN {X 0,Y 375.944,Z 180.653,A -85,B 0,C 180,E1 -12209.685,E2 -12209.685} C_VEL
LIN {X 0,Y 375.972,Z 180.651,A -85,B 0,C 180,E1 -12212.139,E2 -12212.139} C_VEL
LIN {X 0,Y 375.982,Z 180.653,A -85,B 0,C 180,E1 -12214.537,E2 -12214.537} C_VEL
LIN {X 0,Y 375.992,Z 180.649,A -85,B 0,C 180,E1 -12218.047,E2 -12218.047} C_VEL
LIN {X 0,Y 376.003,Z 180.646,A -85,B 0,C 180,E1 -12221.473,E2 -12221.473} C_VEL
LIN {X 0,Y 376.037,Z 180.643,A -85,B 0,C 180,E1 -12224.831,E2 -12224.831} C_VEL
LIN {X 0,Y 376.042,Z 180.646,A -85,B 0,C 180,E1 -12228.136,E2 -12228.136} C_VEL
LIN {X 0,Y 376.234,Z 180.621,A -85,B 0,C 180,E1 -12231.869,E2 -12231.869} C_VEL
LIN {X 0,Y 376.152,Z 180.627,A -85,B 0,C 180,E1 -12234.639,E2 -12234.639} C_VEL
LIN {X 0,Y 376.32,Z 180.611,A -85,B 0,C 180,E1 -12237.859,E2 -12237.859} C_VEL
LIN {X 0,Y 376.453,Z 180.594,A -85,B 0,C 180,E1 -12240,E2 -12240} C_VEL
LIN {X 0,Y 376.19,Z 180.625,A -85,B 0,C 180,E1 -12243.213,E2 -12243.213} C_VEL
LIN {X 0,Y 376.224,Z 180.618,A -85,B 0,C 180,E1 -12246.435,E2 -12246.435} C_VEL
LIN {X 0,Y 376.178,Z 180.624,A -85,B 0,C 180,E1 -12248.596,E2 -12248.596} C_VEL
LIN {X 0,Y 376.031,Z 180.644,A -85,B 0,C 180,E1 -12251.864,E2 -12251.864} C_VEL
LIN {X 0,Y 376.028,Z 180.648,A -85,B 0,C 180,E1 -12255.168,E2 -12255.168} C_VEL
LIN {X 0,Y 376.001,Z 180.647,A -85,B 0,C 180,E1 -12258.527,E2 -12258.527} C_VEL
LIN {X 0,Y 375.991,Z 180.647,A -85,B 0,C 180,E1 -12261.952,E2 -12261.952} C_VEL
LIN {X 0,Y 375.98,Z 180.65,A -85,B 0,C 180,E1 -12265.463,E2 -12265.463} C_VEL
LIN {X 0,Y 375.948,Z 180.656,A -85,B 0,C 180,E1 -12269.081,E2 -12269.081} C_VEL
LIN {X 0,Y 375.925,Z 180.66,A -85,B 0,C 180,E1 -12272.831,E2 -12272.831} C_VEL
LIN {X 0,Y 375.935,Z 180.655,A -85,B 0,C 180,E1 -12275.418,E2 -12275.418} C_VEL
LIN {X 0,Y 375.956,Z 180.655,A -85,B 0,C 180,E1 -12278.273,E2 -12278.273} C_VEL
LIN {X 0,Y 375.97,Z 180.65,A -85,B 0,C 180,E1 -12281.613,E2 -12281.613} C_VEL
LIN {X 0,Y 375.998,Z 180.649,A -85,B 0,C 180,E1 -12285.258,E2 -12285.258} C_VEL
LIN {X 0,Y 376.012,Z 180.73,A -85,B 0,C 180,E1 -12288.234,E2 -12288.234} C_VEL
LIN {X 0,Y 376.842,Z 185.687,A -85,B 0,C 180,E1 -12291.563,E2 -12291.563} C_VEL
LIN {X 0,Y 377.217,Z 189.659,A -85,B 0,C 180,E1 -12294.068,E2 -12294.068} C_VEL
LIN {X 0,Y 376.912,Z 194.67,A -85,B 0,C 180,E1 -12297.043,E2 -12297.043} C_VEL
LIN {X 0,Y 376.439,Z 200.449,A -85,B 0,C 180,E1 -12300.35,E2 -12300.35} C_VEL
LIN {X 0,Y 375.922,Z 206.681,A -85,B 0,C 180,E1 -12303.816,E2 -12303.816} C_VEL
LIN {X 0,Y 375.446,Z 214.413,A -85,B 0,C 180,E1 -12308.016,E2 -12308.016} C_VEL
LIN {X 0,Y 375.106,Z 219.994,A -85,B 0,C 180,E1 -12310.951,E2 -12310.951} C_VEL
LIN {X 0,Y 377.564,Z 233.095,A -85,B 0,C 180,E1 -12311.513,E2 -12311.513} C_VEL
LIN {X 0,Y 379.374,Z 246.354,A -85,B 0,C 180,E1 -12312.288,E2 -12312.288} C_VEL
LIN {X 0,Y 380.104,Z 253.497,A -85,B 0,C 180,E1 -12312.794,E2 -12312.794} C_VEL
LIN {X 0,Y 379.16,Z 265.134,A -85,B 0,C 180,E1 -12313.721,E2 -12313.721} C_VEL
LIN {X 0,Y 378.11,Z 276.847,A -85,B 0,C 180,E1 -12314.919,E2 -12314.919} C_VEL
LIN {X 0,Y 377.193,Z 287.233,A -85,B 0,C 180,E1 -12316.259,E2 -12316.259} C_VEL
LIN {X 0,Y 376.447,Z 295.653,A -85,B 0,C 180,E1 -12317.604,E2 -12317.604} C_VEL
LIN {X 0,Y 375.63,Z 303.881,A -85,B 0,C 180,E1 -12319.218,E2 -12319.218} C_VEL
LIN {X 0,Y 375.174,Z 310.512,A -85,B 0,C 180,E1 -12320.839,E2 -12320.839} C_VEL
LIN {X 0,Y 374.794,Z 315.794,A -85,B 0,C 180,E1 -12322.459,E2 -12322.459} C_VEL
LIN {X 0,Y 374.59,Z 319.538,A -85,B 0,C 180,E1 -12323.923,E2 -12323.923} C_VEL
LIN {X 0,Y 374.551,Z 322.947,A -85,B 0,C 180,E1 -12325.697,E2 -12325.697} C_VEL
LIN {X 0,Y 374.461,Z 324.451,A -85,B 0,C 180,E1 -12326.773,E2 -12326.773} C_VEL
LIN {X 0,Y 374.517,Z 326.173,A -85,B 0,C 180,E1 -12328.926,E2 -12328.926} C_VEL
LIN {X 0,Y 374.554,Z 326.452,A -85,B 0,C 180,E1 -12330.001,E2 -12330.001} C_VEL
LIN {X 0,Y 374.502,Z 326.334,A -85,B 0,C 180,E1 -12331.076,E2 -12331.076} C_VEL
LIN {X 0,Y 374.46,Z 324.844,A -85,B 0,C 180,E1 -12333.228,E2 -12333.228} C_VEL
LIN {X 0,Y 374.529,Z 323.511,A -85,B 0,C 180,E1 -12334.305,E2 -12334.305} C_VEL
LIN {X 0,Y 374.566,Z 320.452,A -85,B 0,C 180,E1 -12336.043,E2 -12336.043} C_VEL
LIN {X 0,Y 374.804,Z 316.846,A -85,B 0,C 180,E1 -12337.542,E2 -12337.542} C_VEL
LIN {X 0,Y 375.198,Z 311.884,A -85,B 0,C 180,E1 -12339.162,E2 -12339.162} C_VEL
LIN {X 0,Y 375.751,Z 305.65,A -85,B 0,C 180,E1 -12340.78,E2 -12340.78} C_VEL
LIN {X 0,Y 376.591,Z 297.876,A -85,B 0,C 180,E1 -12342.393,E2 -12342.393} C_VEL
LIN {X 0,Y 377.6,Z 288.155,A -85,B 0,C 180,E1 -12344.002,E2 -12344.002} C_VEL
LIN {X 0,Y 378.568,Z 278.112,A -85,B 0,C 180,E1 -12345.34,E2 -12345.34} C_VEL
LIN {X 0,Y 379.652,Z 266.742,A -85,B 0,C 180,E1 -12346.535,E2 -12346.535} C_VEL
LIN {X 0,Y 380.7,Z 256.059,A -85,B 0,C 180,E1 -12347.42,E2 -12347.42} C_VEL
LIN {X 0,Y 380.404,Z 249.405,A -85,B 0,C 180,E1 -12347.918,E2 -12347.918} C_VEL
LIN {X 0,Y 378.708,Z 237.127,A -85,B 0,C 180,E1 -12348.712,E2 -12348.712} C_VEL
LIN {X 0,Y 375.991,Z 223.753,A -85,B 0,C 180,E1 -12349.387,E2 -12349.387} C_VEL
LIN {X 0,Y 375.19,Z 219.73,A -85,B 0,C 180,E1 -12349.563,E2 -12349.563} C_VEL
LIN {X 0,Y 375.611,Z 213.125,A -85,B 0,C 180,E1 -12353.136,E2 -12353.136} C_VEL
LIN {X 0,Y 376.054,Z 206.821,A -85,B 0,C 180,E1 -12356.648,E2 -12356.648} C_VEL
LIN {X 0,Y 376.542,Z 201.513,A -85,B 0,C 180,E1 -12359.643,E2 -12359.643} C_VEL
LIN {X 0,Y 377.071,Z 195.718,A -85,B 0,C 180,E1 -12362.994,E2 -12362.994} C_VEL
LIN {X 0,Y 377.369,Z 190.889,A -85,B 0,C 180,E1 -12365.917,E2 -12365.917} C_VEL
LIN {X 0,Y 377.029,Z 186.936,A -85,B 0,C 180,E1 -12368.473,E2 -12368.473} C_VEL
LIN {X 0,Y 376.296,Z 182.294,A -85,B 0,C 180,E1 -12371.663,E2 -12371.663} C_VEL
LIN {X 0,Y 376.006,Z 180.646,A -85,B 0,C 180,E1 -12372.991,E2 -12372.991} C_VEL
LIN {X 0,Y 375.925,Z 180.661,A -85,B 0,C 180,E1 -12376.233,E2 -12376.233} C_VEL
LIN {X 0,Y 375.972,Z 180.651,A -85,B 0,C 180,E1 -12380.028,E2 -12380.028} C_VEL
LIN {X 0,Y 375.948,Z 180.658,A -85,B 0,C 180,E1 -12383.494,E2 -12383.494} C_VEL
LIN {X 0,Y 375.944,Z 180.654,A -85,B 0,C 180,E1 -12385.887,E2 -12385.887} C_VEL
LIN {X 0,Y 375.946,Z 180.654,A -85,B 0,C 180,E1 -12389.686,E2 -12389.686} C_VEL
LIN {X 0,Y 376.001,Z 180.649,A -85,B 0,C 180,E1 -12393.347,E2 -12393.347} C_VEL
LIN {X 0,Y 376.006,Z 180.65,A -85,B 0,C 180,E1 -12396.889,E2 -12396.889} C_VEL
LIN {X 0,Y 375.997,Z 180.647,A -85,B 0,C 180,E1 -12400.339,E2 -12400.339} C_VEL
LIN {X 0,Y 376.009,Z 180.644,A -85,B 0,C 180,E1 -12403.718,E2 -12403.718} C_VEL
LIN {X 0,Y 376.085,Z 180.637,A -85,B 0,C 180,E1 -12407.042,E2 -12407.042} C_VEL
LIN {X 0,Y 376.103,Z 180.637,A -85,B 0,C 180,E1 -12410.318,E2 -12410.318} C_VEL
LIN {X 0,Y 376.242,Z 180.616,A -85,B 0,C 180,E1 -12413.565,E2 -12413.565} C_VEL
LIN {X 0,Y 376.326,Z 180.607,A -85,B 0,C 180,E1 -12417.86,E2 -12417.86} C_VEL
LIN {X 0,Y 376.46,Z 180.592,A -85,B 0,C 180,E1 -12420,E2 -12420} C_VEL
LIN {X 0,Y 376.198,Z 180.621,A -85,B 0,C 180,E1 -12423.213,E2 -12423.213} C_VEL
LIN {X 0,Y 376.212,Z 180.62,A -85,B 0,C 180,E1 -12426.564,E2 -12426.564} C_VEL
LIN {X 0,Y 376.096,Z 180.638,A -85,B 0,C 180,E1 -12429.682,E2 -12429.682} C_VEL
LIN {X 0,Y 376.069,Z 180.642,A -85,B 0,C 180,E1 -12433.658,E2 -12433.658} C_VEL
LIN {X 0,Y 376.035,Z 180.647,A -85,B 0,C 180,E1 -12437.613,E2 -12437.613} C_VEL
LIN {X 0,Y 375.96,Z 180.651,A -85,B 0,C 180,E1 -12440.834,E2 -12440.834} C_VEL
LIN {X 0,Y 375.975,Z 180.649,A -85,B 0,C 180,E1 -12444.283,E2 -12444.283} C_VEL
LIN {X 0,Y 376.003,Z 180.646,A -85,B 0,C 180,E1 -12446.654,E2 -12446.654} C_VEL
LIN {X 0,Y 375.957,Z 180.655,A -85,B 0,C 180,E1 -12449.081,E2 -12449.081} C_VEL
LIN {X 0,Y 375.935,Z 180.657,A -85,B 0,C 180,E1 -12452.83,E2 -12452.83} C_VEL
LIN {X 0,Y 375.943,Z 180.655,A -85,B 0,C 180,E1 -12455.418,E2 -12455.418} C_VEL
LIN {X 0,Y 375.96,Z 180.651,A -85,B 0,C 180,E1 -12458.272,E2 -12458.272} C_VEL
LIN {X 0,Y 375.923,Z 180.655,A -85,B 0,C 180,E1 -12461.602,E2 -12461.602} C_VEL
LIN {X 0,Y 375.918,Z 180.657,A -85,B 0,C 180,E1 -12465.271,E2 -12465.271} C_VEL
LIN {X 0,Y 375.914,Z 180.66,A -85,B 0,C 180,E1 -12468.404,E2 -12468.404} C_VEL
LIN {X 0,Y 375.914,Z 180.662,A -85,B 0,C 180,E1 -12470.534,E2 -12470.534} C_VEL
LIN {X 0,Y 375.928,Z 181.396,A -85,B 0,C 180,E1 -12471.91,E2 -12471.91} C_VEL
LIN {X 0,Y 375.895,Z 184.352,A -85,B 0,C 180,E1 -12474.58,E2 -12474.58} C_VEL
LIN {X 0,Y 375.654,Z 188.783,A -85,B 0,C 180,E1 -12478.411,E2 -12478.411} C_VEL
LIN {X 0,Y 375.41,Z 193.215,A -85,B 0,C 180,E1 -12482.095,E2 -12482.095} C_VEL
LIN {X 0,Y 375.194,Z 197.708,A -85,B 0,C 180,E1 -12485.664,E2 -12485.664} C_VEL
LIN {X 0,Y 375.049,Z 201.516,A -85,B 0,C 180,E1 -12488.523,E2 -12488.523} C_VEL
LIN {X 0,Y 378.599,Z 214.867,A -85,B 0,C 180,E1 -12489.215,E2 -12489.215} C_VEL
LIN {X 0,Y 381.085,Z 226.963,A -85,B 0,C 180,E1 -12490.01,E2 -12490.01} C_VEL
LIN {X 0,Y 381.498,Z 231.854,A -85,B 0,C 180,E1 -12490.362,E2 -12490.362} C_VEL
LIN {X 0,Y 380.628,Z 243.776,A -85,B 0,C 180,E1 -12491.288,E2 -12491.288} C_VEL
LIN {X 0,Y 379.579,Z 254.465,A -85,B 0,C 180,E1 -12492.351,E2 -12492.351} C_VEL
LIN {X 0,Y 378.679,Z 264.197,A -85,B 0,C 180,E1 -12493.559,E2 -12493.559} C_VEL
LIN {X 0,Y 377.654,Z 273.046,A -85,B 0,C 180,E1 -12494.899,E2 -12494.899} C_VEL
LIN {X 0,Y 376.853,Z 280.339,A -85,B 0,C 180,E1 -12496.245,E2 -12496.245} C_VEL
LIN {X 0,Y 376.208,Z 287.506,A -85,B 0,C 180,E1 -12497.868,E2 -12497.868} C_VEL
LIN {X 0,Y 375.564,Z 292.335,A -85,B 0,C 180,E1 -12499.215,E2 -12499.215} C_VEL
LIN {X 0,Y 375.187,Z 297.019,A -85,B 0,C 180,E1 -12500.838,E2 -12500.838} C_VEL
LIN {X 0,Y 374.871,Z 300.597,A -85,B 0,C 180,E1 -12502.459,E2 -12502.459} C_VEL
LIN {X 0,Y 374.7,Z 302.755,A -85,B 0,C 180,E1 -12503.771,E2 -12503.771} C_VEL
LIN {X 0,Y 374.573,Z 304.798,A -85,B 0,C 180,E1 -12505.695,E2 -12505.695} C_VEL
LIN {X 0,Y 374.512,Z 305.608,A -85,B 0,C 180,E1 -12507.849,E2 -12507.849} C_VEL
LIN {X 0,Y 374.544,Z 305.392,A -85,B 0,C 180,E1 -12508.924,E2 -12508.924} C_VEL
LIN {X 0,Y 374.607,Z 303.809,A -85,B 0,C 180,E1 -12511.074,E2 -12511.074} C_VEL
LIN {X 0,Y 374.721,Z 302.432,A -85,B 0,C 180,E1 -12512.149,E2 -12512.149} C_VEL
LIN {X 0,Y 374.969,Z 299.539,A -85,B 0,C 180,E1 -12513.76,E2 -12513.76} C_VEL
LIN {X 0,Y 375.14,Z 295.63,A -85,B 0,C 180,E1 -12515.374,E2 -12515.374} C_VEL
LIN {X 0,Y 375.665,Z 290.017,A -85,B 0,C 180,E1 -12517.142,E2 -12517.142} C_VEL
LIN {X 0,Y 376.249,Z 283.019,A -85,B 0,C 180,E1 -12518.863,E2 -12518.863} C_VEL
LIN {X 0,Y 377.083,Z 274.841,A -85,B 0,C 180,E1 -12520.468,E2 -12520.468} C_VEL
LIN {X 0,Y 377.976,Z 266.459,A -85,B 0,C 180,E1 -12521.8,E2 -12521.8} C_VEL
LIN {X 0,Y 378.869,Z 256.108,A -85,B 0,C 180,E1 -12523.133,E2 -12523.133} C_VEL
LIN {X 0,Y 379.488,Z 247.287,A -85,B 0,C 180,E1 -12524.066,E2 -12524.066} C_VEL
LIN {X 0,Y 380.306,Z 238.156,A -85,B 0,C 180,E1 -12524.855,E2 -12524.855} C_VEL
LIN {X 0,Y 380.665,Z 227.99,A -85,B 0,C 180,E1 -12525.581,E2 -12525.581} C_VEL
LIN {X 0,Y 378.242,Z 214.919,A -85,B 0,C 180,E1 -12526.411,E2 -12526.411} C_VEL
LIN {X 0,Y 375.044,Z 201.293,A -85,B 0,C 180,E1 -12527.074,E2 -12527.074} C_VEL
LIN {X 0,Y 375.189,Z 196.394,A -85,B 0,C 180,E1 -12530.847,E2 -12530.847} C_VEL
LIN {X 0,Y 375.319,Z 193.114,A -85,B 0,C 180,E1 -12533.429,E2 -12533.429} C_VEL
LIN {X 0,Y 375.376,Z 190.88,A -85,B 0,C 180,E1 -12535.205,E2 -12535.205} C_VEL
LIN {X 0,Y 374.804,Z 189.874,A -85,B 0,C 180,E1 -12536.088,E2 -12536.088} C_VEL
LIN {X 0,Y 372.056,Z 188.473,A -85,B 0,C 180,E1 -12537.532,E2 -12537.532} C_VEL
LIN {X 0,Y 369.696,Z 187.405,A -85,B 0,C 180,E1 -12538.702,E2 -12538.702} C_VEL
LIN {X 0,Y 368.696,Z 186.492,A -85,B 0,C 180,E1 -12539.602,E2 -12539.602} C_VEL
LIN {X 0,Y 368.624,Z 186.151,A -85,B 0,C 180,E1 -12539.906,E2 -12539.906} C_VEL
LIN {X 0,Y 368.779,Z 182.605,A -85,B 0,C 180,E1 -12543.014,E2 -12543.014} C_VEL
LIN {X 0,Y 368.749,Z 182.023,A -85,B 0,C 180,E1 -12543.55,E2 -12543.55} C_VEL
LIN {X 0,Y 368.841,Z 181.541,A -85,B 0,C 180,E1 -12544.981,E2 -12544.981} C_VEL
LIN {X 0,Y 368.888,Z 181.537,A -85,B 0,C 180,E1 -12547.561,E2 -12547.561} C_VEL
LIN {X 0,Y 368.898,Z 181.531,A -85,B 0,C 180,E1 -12550.367,E2 -12550.367} C_VEL
LIN {X 0,Y 368.875,Z 181.536,A -85,B 0,C 180,E1 -12553.614,E2 -12553.614} C_VEL
LIN {X 0,Y 368.923,Z 181.529,A -85,B 0,C 180,E1 -12556.701,E2 -12556.701} C_VEL
LIN {X 0,Y 368.936,Z 181.527,A -85,B 0,C 180,E1 -12559.633,E2 -12559.633} C_VEL
LIN {X 0,Y 368.882,Z 181.537,A -85,B 0,C 180,E1 -12563.142,E2 -12563.142} C_VEL
LIN {X 0,Y 368.875,Z 181.536,A -85,B 0,C 180,E1 -12566.459,E2 -12566.459} C_VEL
LIN {X 0,Y 368.907,Z 181.533,A -85,B 0,C 180,E1 -12569.044,E2 -12569.044} C_VEL
LIN {X 0,Y 368.957,Z 181.523,A -85,B 0,C 180,E1 -12571.562,E2 -12571.562} C_VEL
LIN {X 0,Y 368.936,Z 181.526,A -85,B 0,C 180,E1 -12575.223,E2 -12575.223} C_VEL
LIN {X 0,Y 368.948,Z 181.526,A -85,B 0,C 180,E1 -12578.956,E2 -12578.956} C_VEL
LIN {X 0,Y 368.964,Z 181.528,A -85,B 0,C 180,E1 -12582.255,E2 -12582.255} C_VEL
LIN {X 0,Y 368.99,Z 181.52,A -85,B 0,C 180,E1 -12585.664,E2 -12585.664} C_VEL
LIN {X 0,Y 369.023,Z 181.515,A -85,B 0,C 180,E1 -12589.021,E2 -12589.021} C_VEL
LIN {X 0,Y 369.172,Z 181.499,A -85,B 0,C 180,E1 -12592.342,E2 -12592.342} C_VEL
LIN {X 0,Y 369.125,Z 181.503,A -85,B 0,C 180,E1 -12594.537,E2 -12594.537} C_VEL
LIN {X 0,Y 369.285,Z 181.488,A -85,B 0,C 180,E1 -12597.818,E2 -12597.818} C_VEL
LIN {X 0,Y 369.423,Z 181.469,A -85,B 0,C 180,E1 -12600,E2 -12600} C_VEL
LIN {X 0,Y 369.128,Z 181.504,A -85,B 0,C 180,E1 -12603.274,E2 -12603.274} C_VEL
LIN {X 0,Y 369.184,Z 181.495,A -85,B 0,C 180,E1 -12606.558,E2 -12606.558} C_VEL
LIN {X 0,Y 369.112,Z 181.504,A -85,B 0,C 180,E1 -12608.761,E2 -12608.761} C_VEL
LIN {X 0,Y 368.984,Z 181.52,A -85,B 0,C 180,E1 -12612.094,E2 -12612.094} C_VEL
LIN {X 0,Y 368.967,Z 181.526,A -85,B 0,C 180,E1 -12615.466,E2 -12615.466} C_VEL
LIN {X 0,Y 368.963,Z 181.526,A -85,B 0,C 180,E1 -12618.894,E2 -12618.894} C_VEL
LIN {X 0,Y 368.946,Z 181.525,A -85,B 0,C 180,E1 -12622.394,E2 -12622.394} C_VEL
LIN {X 0,Y 368.974,Z 181.521,A -85,B 0,C 180,E1 -12625.982,E2 -12625.982} C_VEL
LIN {X 0,Y 368.937,Z 181.532,A -85,B 0,C 180,E1 -12628.814,E2 -12628.814} C_VEL
LIN {X 0,Y 368.874,Z 181.535,A -85,B 0,C 180,E1 -12632.24,E2 -12632.24} C_VEL
LIN {X 0,Y 368.906,Z 181.532,A -85,B 0,C 180,E1 -12635.004,E2 -12635.004} C_VEL
LIN {X 0,Y 368.892,Z 181.536,A -85,B 0,C 180,E1 -12638.643,E2 -12638.643} C_VEL
LIN {X 0,Y 368.923,Z 181.53,A -85,B 0,C 180,E1 -12642.022,E2 -12642.022} C_VEL
LIN {X 0,Y 368.973,Z 181.524,A -85,B 0,C 180,E1 -12645.195,E2 -12645.195} C_VEL
LIN {X 0,Y 368.979,Z 181.618,A -85,B 0,C 180,E1 -12647.974,E2 -12647.974} C_VEL
LIN {X 0,Y 369.762,Z 186.312,A -85,B 0,C 180,E1 -12651.195,E2 -12651.195} C_VEL
LIN {X 0,Y 370.207,Z 190.569,A -85,B 0,C 180,E1 -12653.953,E2 -12653.953} C_VEL
LIN {X 0,Y 369.936,Z 195.108,A -85,B 0,C 180,E1 -12656.711,E2 -12656.711} C_VEL
LIN {X 0,Y 369.392,Z 201.337,A -85,B 0,C 180,E1 -12660.355,E2 -12660.355} C_VEL
LIN {X 0,Y 368.833,Z 207.779,A -85,B 0,C 180,E1 -12664.01,E2 -12664.01} C_VEL
LIN {X 0,Y 368.342,Z 215.255,A -85,B 0,C 180,E1 -12668.16,E2 -12668.16} C_VEL
LIN {X 0,Y 368.055,Z 219.816,A -85,B 0,C 180,E1 -12670.589,E2 -12670.589} C_VEL
LIN {X 0,Y 370.575,Z 233.119,A -85,B 0,C 180,E1 -12671.179,E2 -12671.179} C_VEL
LIN {X 0,Y 372.324,Z 245.071,A -85,B 0,C 180,E1 -12671.89,E2 -12671.89} C_VEL
LIN {X 0,Y 373.202,Z 254.929,A -85,B 0,C 180,E1 -12672.607,E2 -12672.607} C_VEL
LIN {X 0,Y 372.21,Z 266.204,A -85,B 0,C 180,E1 -12673.549,E2 -12673.549} C_VEL
LIN {X 0,Y 371.125,Z 277.637,A -85,B 0,C 180,E1 -12674.762,E2 -12674.762} C_VEL
LIN {X 0,Y 370.275,Z 286.932,A -85,B 0,C 180,E1 -12675.997,E2 -12675.997} C_VEL
LIN {X 0,Y 369.48,Z 295.37,A -85,B 0,C 180,E1 -12677.366,E2 -12677.366} C_VEL
LIN {X 0,Y 368.61,Z 303.612,A -85,B 0,C 180,E1 -12679.01,E2 -12679.01} C_VEL
LIN {X 0,Y 368.106,Z 310.255,A -85,B 0,C 180,E1 -12680.662,E2 -12680.662} C_VEL
LIN {X 0,Y 367.717,Z 315.549,A -85,B 0,C 180,E1 -12682.313,E2 -12682.313} C_VEL
LIN {X 0,Y 367.507,Z 319.622,A -85,B 0,C 180,E1 -12683.945,E2 -12683.945} C_VEL
LIN {X 0,Y 367.457,Z 322.724,A -85,B 0,C 180,E1 -12685.613,E2 -12685.613} C_VEL
LIN {X 0,Y 367.38,Z 324.236,A -85,B 0,C 180,E1 -12686.711,E2 -12686.711} C_VEL
LIN {X 0,Y 367.417,Z 325.968,A -85,B 0,C 180,E1 -12688.905,E2 -12688.905} C_VEL
LIN {X 0,Y 367.456,Z 326.252,A -85,B 0,C 180,E1 -12690.001,E2 -12690.001} C_VEL
LIN {X 0,Y 367.402,Z 326.141,A -85,B 0,C 180,E1 -12691.097,E2 -12691.097} C_VEL
LIN {X 0,Y 367.377,Z 324.662,A -85,B 0,C 180,E1 -12693.291,E2 -12693.291} C_VEL
LIN {X 0,Y 367.436,Z 323.333,A -85,B 0,C 180,E1 -12694.388,E2 -12694.388} C_VEL
LIN {X 0,Y 367.475,Z 320.581,A -85,B 0,C 180,E1 -12696.007,E2 -12696.007} C_VEL
LIN {X 0,Y 367.73,Z 316.688,A -85,B 0,C 180,E1 -12697.688,E2 -12697.688} C_VEL
LIN {X 0,Y 368.147,Z 311.736,A -85,B 0,C 180,E1 -12699.339,E2 -12699.339} C_VEL
LIN {X 0,Y 368.732,Z 305.514,A -85,B 0,C 180,E1 -12700.988,E2 -12700.988} C_VEL
LIN {X 0,Y 369.64,Z 297.762,A -85,B 0,C 180,E1 -12702.63,E2 -12702.63} C_VEL
LIN {X 0,Y 370.689,Z 288.059,A -85,B 0,C 180,E1 -12704.268,E2 -12704.268} C_VEL
LIN {X 0,Y 371.584,Z 279.119,A -85,B 0,C 180,E1 -12705.495,E2 -12705.495} C_VEL
LIN {X 0,Y 372.723,Z 268.133,A -85,B 0,C 180,E1 -12706.711,E2 -12706.711} C_VEL
LIN {X 0,Y 373.919,Z 256.15,A -85,B 0,C 180,E1 -12707.74,E2 -12707.74} C_VEL
LIN {X 0,Y 373.369,Z 248.199,A -85,B 0,C 180,E1 -12708.353,E2 -12708.353} C_VEL
LIN {X 0,Y 371.388,Z 235.174,A -85,B 0,C 180,E1 -12709.195,E2 -12709.195} C_VEL
LIN {X 0,Y 368.589,Z 221.79,A -85,B 0,C 180,E1 -12709.867,E2 -12709.867} C_VEL
LIN {X 0,Y 368.143,Z 219.521,A -85,B 0,C 180,E1 -12709.97,E2 -12709.97} C_VEL
LIN {X 0,Y 368.545,Z 214.049,A -85,B 0,C 180,E1 -12713.011,E2 -12713.011} C_VEL
LIN {X 0,Y 368.955,Z 207.956,A -85,B 0,C 180,E1 -12716.456,E2 -12716.456} C_VEL
LIN {X 0,Y 369.511,Z 202.461,A -85,B 0,C 180,E1 -12719.636,E2 -12719.636} C_VEL
LIN {X 0,Y 369.897,Z 198.197,A -85,B 0,C 180,E1 -12722.139,E2 -12722.139} C_VEL
LIN {X 0,Y 370.294,Z 193.957,A -85,B 0,C 180,E1 -12724.705,E2 -12724.705} C_VEL
LIN {X 0,Y 370.238,Z 190.155,A -85,B 0,C 180,E1 -12727.131,E2 -12727.131} C_VEL
LIN {X 0,Y 369.649,Z 185.549,A -85,B 0,C 180,E1 -12730.27,E2 -12730.27} C_VEL
LIN {X 0,Y 368.931,Z 181.528,A -85,B 0,C 180,E1 -12733.295,E2 -12733.295} C_VEL
LIN {X 0,Y 368.878,Z 181.542,A -85,B 0,C 180,E1 -12736.695,E2 -12736.695} C_VEL
LIN {X 0,Y 368.897,Z 181.535,A -85,B 0,C 180,E1 -12739.642,E2 -12739.642} C_VEL
LIN {X 0,Y 368.886,Z 181.535,A -85,B 0,C 180,E1 -12743.143,E2 -12743.143} C_VEL
LIN {X 0,Y 368.881,Z 181.532,A -85,B 0,C 180,E1 -12746.46,E2 -12746.46} C_VEL
LIN {X 0,Y 368.896,Z 181.53,A -85,B 0,C 180,E1 -12750.308,E2 -12750.308} C_VEL
LIN {X 0,Y 368.982,Z 181.52,A -85,B 0,C 180,E1 -12754.019,E2 -12754.019} C_VEL
LIN {X 0,Y 368.954,Z 181.524,A -85,B 0,C 180,E1 -12757.606,E2 -12757.606} C_VEL
LIN {X 0,Y 368.973,Z 181.524,A -85,B 0,C 180,E1 -12761.107,E2 -12761.107} C_VEL
LIN {X 0,Y 368.978,Z 181.524,A -85,B 0,C 180,E1 -12764.535,E2 -12764.535} C_VEL
LIN {X 0,Y 368.991,Z 181.519,A -85,B 0,C 180,E1 -12767.906,E2 -12767.906} C_VEL
LIN {X 0,Y 369.154,Z 181.499,A -85,B 0,C 180,E1 -12771.859,E2 -12771.859} C_VEL
LIN {X 0,Y 369.133,Z 181.506,A -85,B 0,C 180,E1 -12774.538,E2 -12774.538} C_VEL
LIN {X 0,Y 369.292,Z 181.483,A -85,B 0,C 180,E1 -12777.819,E2 -12777.819} C_VEL
LIN {X 0,Y 369.409,Z 181.47,A -85,B 0,C 180,E1 -12780,E2 -12780} C_VEL
LIN {X 0,Y 369.301,Z 181.486,A -85,B 0,C 180,E1 -12782.182,E2 -12782.182} C_VEL
LIN {X 0,Y 369.183,Z 181.496,A -85,B 0,C 180,E1 -12786.559,E2 -12786.559} C_VEL
LIN {X 0,Y 369.045,Z 181.518,A -85,B 0,C 180,E1 -12789.869,E2 -12789.869} C_VEL
LIN {X 0,Y 369.017,Z 181.522,A -85,B 0,C 180,E1 -12793.773,E2 -12793.773} C_VEL
LIN {X 0,Y 368.98,Z 181.525,A -85,B 0,C 180,E1 -12797.744,E2 -12797.744} C_VEL
LIN {X 0,Y 368.911,Z 181.532,A -85,B 0,C 180,E1 -12801.221,E2 -12801.221} C_VEL
LIN {X 0,Y 368.94,Z 181.526,A -85,B 0,C 180,E1 -12804.777,E2 -12804.777} C_VEL
LIN {X 0,Y 368.952,Z 181.528,A -85,B 0,C 180,E1 -12807.205,E2 -12807.205} C_VEL
LIN {X 0,Y 368.906,Z 181.531,A -85,B 0,C 180,E1 -12809.692,E2 -12809.692} C_VEL
LIN {X 0,Y 368.883,Z 181.537,A -85,B 0,C 180,E1 -12813.045,E2 -12813.045} C_VEL
LIN {X 0,Y 368.904,Z 181.53,A -85,B 0,C 180,E1 -12816.199,E2 -12816.199} C_VEL
LIN {X 0,Y 368.89,Z 181.537,A -85,B 0,C 180,E1 -12818.955,E2 -12818.955} C_VEL
LIN {X 0,Y 368.87,Z 181.534,A -85,B 0,C 180,E1 -12822.011,E2 -12822.011} C_VEL
LIN {X 0,Y 368.871,Z 181.535,A -85,B 0,C 180,E1 -12825.177,E2 -12825.177} C_VEL
LIN {X 0,Y 368.865,Z 181.536,A -85,B 0,C 180,E1 -12828.178,E2 -12828.178} C_VEL
LIN {X 0,Y 368.845,Z 181.544,A -85,B 0,C 180,E1 -12831.042,E2 -12831.042} C_VEL
LIN {X 0,Y 368.907,Z 184.477,A -85,B 0,C 180,E1 -12833.804,E2 -12833.804} C_VEL
LIN {X 0,Y 368.692,Z 188.061,A -85,B 0,C 180,E1 -12837.007,E2 -12837.007} C_VEL
LIN {X 0,Y 368.47,Z 191.865,A -85,B 0,C 180,E1 -12840.272,E2 -12840.272} C_VEL
LIN {X 0,Y 368.266,Z 196.357,A -85,B 0,C 180,E1 -12843.965,E2 -12843.965} C_VEL
LIN {X 0,Y 368.013,Z 200.842,A -85,B 0,C 180,E1 -12847.547,E2 -12847.547} C_VEL
LIN {X 0,Y 367.984,Z 201.558,A -85,B 0,C 180,E1 -12848.106,E2 -12848.106} C_VEL
LIN {X 0,Y 371.667,Z 215.22,A -85,B 0,C 180,E1 -12848.84,E2 -12848.84} C_VEL
LIN {X 0,Y 374.086,Z 227.137,A -85,B 0,C 180,E1 -12849.641,E2 -12849.641} C_VEL
LIN {X 0,Y 374.79,Z 231.895,A -85,B 0,C 180,E1 -12850.007,E2 -12850.007} C_VEL
LIN {X 0,Y 373.904,Z 243.729,A -85,B 0,C 180,E1 -12850.939,E2 -12850.939} C_VEL
LIN {X 0,Y 372.819,Z 254.474,A -85,B 0,C 180,E1 -12852.021,E2 -12852.021} C_VEL
LIN {X 0,Y 371.847,Z 264.238,A -85,B 0,C 180,E1 -12853.249,E2 -12853.249} C_VEL
LIN {X 0,Y 370.766,Z 273.113,A -85,B 0,C 180,E1 -12854.611,E2 -12854.611} C_VEL
LIN {X 0,Y 369.893,Z 280.446,A -85,B 0,C 180,E1 -12855.985,E2 -12855.985} C_VEL
LIN {X 0,Y 369.258,Z 287.615,A -85,B 0,C 180,E1 -12857.636,E2 -12857.636} C_VEL
LIN {X 0,Y 368.55,Z 292.46,A -85,B 0,C 180,E1 -12859.007,E2 -12859.007} C_VEL
LIN {X 0,Y 368.163,Z 297.159,A -85,B 0,C 180,E1 -12860.662,E2 -12860.662} C_VEL
LIN {X 0,Y 367.814,Z 300.752,A -85,B 0,C 180,E1 -12862.313,E2 -12862.313} C_VEL
LIN {X 0,Y 367.599,Z 303.141,A -85,B 0,C 180,E1 -12863.815,E2 -12863.815} C_VEL
LIN {X 0,Y 367.503,Z 304.979,A -85,B 0,C 180,E1 -12865.612,E2 -12865.612} C_VEL
LIN {X 0,Y 367.413,Z 305.805,A -85,B 0,C 180,E1 -12867.807,E2 -12867.807} C_VEL
LIN {X 0,Y 367.445,Z 305.6,A -85,B 0,C 180,E1 -12868.903,E2 -12868.903} C_VEL
LIN {X 0,Y 367.512,Z 304.029,A -85,B 0,C 180,E1 -12871.095,E2 -12871.095} C_VEL
LIN {X 0,Y 367.629,Z 302.662,A -85,B 0,C 180,E1 -12872.19,E2 -12872.19} C_VEL
LIN {X 0,Y 367.877,Z 299.781,A -85,B 0,C 180,E1 -12873.833,E2 -12873.833} C_VEL
LIN {X 0,Y 368.095,Z 295.885,A -85,B 0,C 180,E1 -12875.477,E2 -12875.477} C_VEL
LIN {X 0,Y 368.601,Z 290.702,A -85,B 0,C 180,E1 -12877.165,E2 -12877.165} C_VEL
LIN {X 0,Y 369.139,Z 284.538,A -85,B 0,C 180,E1 -12878.76,E2 -12878.76} C_VEL
LIN {X 0,Y 369.935,Z 276.635,A -85,B 0,C 180,E1 -12880.396,E2 -12880.396} C_VEL
LIN {X 0,Y 371.048,Z 266.803,A -85,B 0,C 180,E1 -12882.024,E2 -12882.024} C_VEL
LIN {X 0,Y 371.979,Z 256.494,A -85,B 0,C 180,E1 -12883.38,E2 -12883.38} C_VEL
LIN {X 0,Y 372.631,Z 247.712,A -85,B 0,C 180,E1 -12884.33,E2 -12884.33} C_VEL
LIN {X 0,Y 373.486,Z 238.634,A -85,B 0,C 180,E1 -12885.133,E2 -12885.133} C_VEL
LIN {X 0,Y 373.948,Z 229.909,A -85,B 0,C 180,E1 -12885.772,E2 -12885.772} C_VEL
LIN {X 0,Y 371.724,Z 217.363,A -85,B 0,C 180,E1 -12886.624,E2 -12886.624} C_VEL
LIN {X 0,Y 368.653,Z 204.382,A -85,B 0,C 180,E1 -12887.305,E2 -12887.305} C_VEL
LIN {X 0,Y 367.985,Z 201.467,A -85,B 0,C 180,E1 -12887.457,E2 -12887.457} C_VEL
LIN {X 0,Y 368.138,Z 196.622,A -85,B 0,C 180,E1 -12891.265,E2 -12891.265} C_VEL
LIN {X 0,Y 368.312,Z 192.177,A -85,B 0,C 180,E1 -12894.819,E2 -12894.819} C_VEL
LIN {X 0,Y 368.461,Z 189.255,A -85,B 0,C 180,E1 -12897.241,E2 -12897.241} C_VEL
LIN {X 0,Y 368.624,Z 186.151,A -85,B 0,C 180,E1 -12899.906,E2 -12899.906} C_VEL
LIN {X 0,Y 367.979,Z 185.213,A -85,B 0,C 180,E1 -12900.807,E2 -12900.807} C_VEL
LIN {X 0,Y 365.143,Z 183.921,A -85,B 0,C 180,E1 -12902.278,E2 -12902.278} C_VEL
LIN {X 0,Y 362.762,Z 182.935,A -85,B 0,C 180,E1 -12903.474,E2 -12903.474} C_VEL
LIN {X 0,Y 361.787,Z 182.468,A -85,B 0,C 180,E1 -12904.402,E2 -12904.402} C_VEL
LIN {X 0,Y 361.734,Z 182.426,A -85,B 0,C 180,E1 -12904.716,E2 -12904.716} C_VEL
LIN {X 0,Y 361.847,Z 182.412,A -85,B 0,C 180,E1 -12907.218,E2 -12907.218} C_VEL
LIN {X 0,Y 361.823,Z 182.413,A -85,B 0,C 180,E1 -12910.752,E2 -12910.752} C_VEL
LIN {X 0,Y 361.832,Z 182.41,A -85,B 0,C 180,E1 -12914.361,E2 -12914.361} C_VEL
LIN {X 0,Y 361.867,Z 182.408,A -85,B 0,C 180,E1 -12917.557,E2 -12917.557} C_VEL
LIN {X 0,Y 361.855,Z 182.413,A -85,B 0,C 180,E1 -12920.97,E2 -12920.97} C_VEL
LIN {X 0,Y 361.854,Z 182.411,A -85,B 0,C 180,E1 -12924.653,E2 -12924.653} C_VEL
LIN {X 0,Y 361.816,Z 182.415,A -85,B 0,C 180,E1 -12928.368,E2 -12928.368} C_VEL
LIN {X 0,Y 361.878,Z 182.408,A -85,B 0,C 180,E1 -12930.953,E2 -12930.953} C_VEL
LIN {X 0,Y 361.93,Z 182.398,A -85,B 0,C 180,E1 -12933.473,E2 -12933.473} C_VEL
LIN {X 0,Y 361.893,Z 182.404,A -85,B 0,C 180,E1 -12937.144,E2 -12937.144} C_VEL
LIN {X 0,Y 361.907,Z 182.404,A -85,B 0,C 180,E1 -12940.723,E2 -12940.723} C_VEL
LIN {X 0,Y 361.923,Z 182.405,A -85,B 0,C 180,E1 -12944.225,E2 -12944.225} C_VEL
LIN {X 0,Y 361.945,Z 182.398,A -85,B 0,C 180,E1 -12947.667,E2 -12947.667} C_VEL
LIN {X 0,Y 362.141,Z 182.375,A -85,B 0,C 180,E1 -12951.754,E2 -12951.754} C_VEL
LIN {X 0,Y 362.099,Z 182.379,A -85,B 0,C 180,E1 -12954.431,E2 -12954.431} C_VEL
LIN {X 0,Y 362.25,Z 182.364,A -85,B 0,C 180,E1 -12957.776,E2 -12957.776} C_VEL
LIN {X 0,Y 362.372,Z 182.347,A -85,B 0,C 180,E1 -12960,E2 -12960} C_VEL
LIN {X 0,Y 362.258,Z 182.359,A -85,B 0,C 180,E1 -12962.223,E2 -12962.223} C_VEL
LIN {X 0,Y 362.147,Z 182.371,A -85,B 0,C 180,E1 -12966.686,E2 -12966.686} C_VEL
LIN {X 0,Y 362.049,Z 182.385,A -85,B 0,C 180,E1 -12968.934,E2 -12968.934} C_VEL
LIN {X 0,Y 361.938,Z 182.397,A -85,B 0,C 180,E1 -12972.333,E2 -12972.333} C_VEL
LIN {X 0,Y 361.932,Z 182.399,A -85,B 0,C 180,E1 -12974.621,E2 -12974.621} C_VEL
LIN {X 0,Y 361.933,Z 182.398,A -85,B 0,C 180,E1 -12978.101,E2 -12978.101} C_VEL
LIN {X 0,Y 361.897,Z 182.403,A -85,B 0,C 180,E1 -12981.652,E2 -12981.652} C_VEL
LIN {X 0,Y 361.903,Z 182.404,A -85,B 0,C 180,E1 -12985.292,E2 -12985.292} C_VEL
LIN {X 0,Y 361.893,Z 182.403,A -85,B 0,C 180,E1 -12987.78,E2 -12987.78} C_VEL
LIN {X 0,Y 361.823,Z 182.413,A -85,B 0,C 180,E1 -12991.287,E2 -12991.287} C_VEL
LIN {X 0,Y 361.831,Z 182.413,A -85,B 0,C 180,E1 -12994.283,E2 -12994.283} C_VEL
LIN {X 0,Y 361.844,Z 182.41,A -85,B 0,C 180,E1 -12997.225,E2 -12997.225} C_VEL
LIN {X 0,Y 361.886,Z 182.407,A -85,B 0,C 180,E1 -13000.771,E2 -13000.771} C_VEL
LIN {X 0,Y 361.915,Z 182.406,A -85,B 0,C 180,E1 -13004.353,E2 -13004.353} C_VEL
LIN {X 0,Y 361.944,Z 182.418,A -85,B 0,C 180,E1 -13007.641,E2 -13007.641} C_VEL
LIN {X 0,Y 362.681,Z 186.93,A -85,B 0,C 180,E1 -13010.816,E2 -13010.816} C_VEL
LIN {X 0,Y 363.112,Z 190.4,A -85,B 0,C 180,E1 -13013.134,E2 -13013.134} C_VEL
LIN {X 0,Y 363.115,Z 193.626,A -85,B 0,C 180,E1 -13015.186,E2 -13015.186} C_VEL
LIN {X 0,Y 362.617,Z 199.104,A -85,B 0,C 180,E1 -13018.515,E2 -13018.515} C_VEL
LIN {X 0,Y 362.097,Z 204.368,A -85,B 0,C 180,E1 -13021.61,E2 -13021.61} C_VEL
LIN {X 0,Y 361.576,Z 210.778,A -85,B 0,C 180,E1 -13025.301,E2 -13025.301} C_VEL
LIN {X 0,Y 361.131,Z 217.481,A -85,B 0,C 180,E1 -13029.088,E2 -13029.088} C_VEL
LIN {X 0,Y 360.996,Z 219.452,A -85,B 0,C 180,E1 -13030.194,E2 -13030.194} C_VEL
LIN {X 0,Y 363.759,Z 234.073,A -85,B 0,C 180,E1 -13030.885,E2 -13030.885} C_VEL
LIN {X 0,Y 365.601,Z 247.218,A -85,B 0,C 180,E1 -13031.712,E2 -13031.712} C_VEL
LIN {X 0,Y 366.28,Z 256.299,A -85,B 0,C 180,E1 -13032.412,E2 -13032.412} C_VEL
LIN {X 0,Y 365.242,Z 267.272,A -85,B 0,C 180,E1 -13033.37,E2 -13033.37} C_VEL
LIN {X 0,Y 364.185,Z 278.061,A -85,B 0,C 180,E1 -13034.56,E2 -13034.56} C_VEL
LIN {X 0,Y 363.16,Z 288.422,A -85,B 0,C 180,E1 -13036.003,E2 -13036.003} C_VEL
LIN {X 0,Y 362.361,Z 296.579,A -85,B 0,C 180,E1 -13037.399,E2 -13037.399} C_VEL
LIN {X 0,Y 361.512,Z 304.581,A -85,B 0,C 180,E1 -13039.075,E2 -13039.075} C_VEL
LIN {X 0,Y 361.055,Z 309.998,A -85,B 0,C 180,E1 -13040.478,E2 -13040.478} C_VEL
LIN {X 0,Y 360.667,Z 315.305,A -85,B 0,C 180,E1 -13042.162,E2 -13042.162} C_VEL
LIN {X 0,Y 360.433,Z 319.674,A -85,B 0,C 180,E1 -13043.954,E2 -13043.954} C_VEL
LIN {X 0,Y 360.366,Z 322.5,A -85,B 0,C 180,E1 -13045.527,E2 -13045.527} C_VEL
LIN {X 0,Y 360.3,Z 324.021,A -85,B 0,C 180,E1 -13046.646,E2 -13046.646} C_VEL
LIN {X 0,Y 360.316,Z 325.763,A -85,B 0,C 180,E1 -13048.883,E2 -13048.883} C_VEL
LIN {X 0,Y 360.359,Z 326.052,A -85,B 0,C 180,E1 -13050.001,E2 -13050.001} C_VEL
LIN {X 0,Y 360.302,Z 325.948,A -85,B 0,C 180,E1 -13051.118,E2 -13051.118} C_VEL
LIN {X 0,Y 360.297,Z 324.48,A -85,B 0,C 180,E1 -13053.355,E2 -13053.355} C_VEL
LIN {X 0,Y 360.347,Z 323.156,A -85,B 0,C 180,E1 -13054.475,E2 -13054.475} C_VEL
LIN {X 0,Y 360.377,Z 320.727,A -85,B 0,C 180,E1 -13055.961,E2 -13055.961} C_VEL
LIN {X 0,Y 360.68,Z 316.531,A -85,B 0,C 180,E1 -13057.84,E2 -13057.84} C_VEL
LIN {X 0,Y 361.099,Z 311.589,A -85,B 0,C 180,E1 -13059.523,E2 -13059.523} C_VEL
LIN {X 0,Y 361.715,Z 305.38,A -85,B 0,C 180,E1 -13061.204,E2 -13061.204} C_VEL
LIN {X 0,Y 362.684,Z 297.649,A -85,B 0,C 180,E1 -13062.876,E2 -13062.876} C_VEL
LIN {X 0,Y 363.572,Z 289.747,A -85,B 0,C 180,E1 -13064.268,E2 -13064.268} C_VEL
LIN {X 0,Y 364.596,Z 280.114,A -85,B 0,C 180,E1 -13065.656,E2 -13065.656} C_VEL
LIN {X 0,Y 365.783,Z 269.43,A -85,B 0,C 180,E1 -13066.894,E2 -13066.894} C_VEL
LIN {X 0,Y 367.044,Z 257.695,A -85,B 0,C 180,E1 -13067.958,E2 -13067.958} C_VEL
LIN {X 0,Y 366.664,Z 250.052,A -85,B 0,C 180,E1 -13068.571,E2 -13068.571} C_VEL
LIN {X 0,Y 365.057,Z 238.512,A -85,B 0,C 180,E1 -13069.38,E2 -13069.38} C_VEL
LIN {X 0,Y 362.472,Z 225.43,A -85,B 0,C 180,E1 -13070.108,E2 -13070.108} C_VEL
LIN {X 0,Y 361.12,Z 219.311,A -85,B 0,C 180,E1 -13070.414,E2 -13070.414} C_VEL
LIN {X 0,Y 361.45,Z 214.939,A -85,B 0,C 180,E1 -13072.884,E2 -13072.884} C_VEL
LIN {X 0,Y 361.82,Z 209.689,A -85,B 0,C 180,E1 -13075.914,E2 -13075.914} C_VEL
LIN {X 0,Y 362.407,Z 204.071,A -85,B 0,C 180,E1 -13079.23,E2 -13079.23} C_VEL
LIN {X 0,Y 362.867,Z 199.147,A -85,B 0,C 180,E1 -13082.181,E2 -13082.181} C_VEL
LIN {X 0,Y 363.287,Z 194.92,A -85,B 0,C 180,E1 -13084.797,E2 -13084.797} C_VEL
LIN {X 0,Y 363.181,Z 190.798,A -85,B 0,C 180,E1 -13087.495,E2 -13087.495} C_VEL
LIN {X 0,Y 362.779,Z 187.556,A -85,B 0,C 180,E1 -13089.737,E2 -13089.737} C_VEL
LIN {X 0,Y 361.915,Z 182.404,A -85,B 0,C 180,E1 -13093.577,E2 -13093.577} C_VEL
LIN {X 0,Y 361.825,Z 182.417,A -85,B 0,C 180,E1 -13097.567,E2 -13097.567} C_VEL
LIN {X 0,Y 361.852,Z 182.409,A -85,B 0,C 180,E1 -13100.973,E2 -13100.973} C_VEL
LIN {X 0,Y 361.859,Z 182.408,A -85,B 0,C 180,E1 -13104.654,E2 -13104.654} C_VEL
LIN {X 0,Y 361.818,Z 182.412,A -85,B 0,C 180,E1 -13108.369,E2 -13108.369} C_VEL
LIN {X 0,Y 361.889,Z 182.403,A -85,B 0,C 180,E1 -13112.219,E2 -13112.219} C_VEL
LIN {X 0,Y 361.912,Z 182.403,A -85,B 0,C 180,E1 -13114.709,E2 -13114.709} C_VEL
LIN {X 0,Y 361.906,Z 182.402,A -85,B 0,C 180,E1 -13118.348,E2 -13118.348} C_VEL
LIN {X 0,Y 361.949,Z 182.396,A -85,B 0,C 180,E1 -13122.06,E2 -13122.06} C_VEL
LIN {X 0,Y 361.978,Z 182.393,A -85,B 0,C 180,E1 -13126.101,E2 -13126.101} C_VEL
LIN {X 0,Y 362.015,Z 182.388,A -85,B 0,C 180,E1 -13129.938,E2 -13129.938} C_VEL
LIN {X 0,Y 362.161,Z 182.369,A -85,B 0,C 180,E1 -13133.314,E2 -13133.314} C_VEL
LIN {X 0,Y 362.256,Z 182.359,A -85,B 0,C 180,E1 -13137.777,E2 -13137.777} C_VEL
LIN {X 0,Y 362.36,Z 182.349,A -85,B 0,C 180,E1 -13140,E2 -13140} C_VEL
LIN {X 0,Y 362.267,Z 182.362,A -85,B 0,C 180,E1 -13142.224,E2 -13142.224} C_VEL
LIN {X 0,Y 362.144,Z 182.372,A -85,B 0,C 180,E1 -13146.687,E2 -13146.687} C_VEL
LIN {X 0,Y 361.98,Z 182.396,A -85,B 0,C 180,E1 -13150.064,E2 -13150.064} C_VEL
LIN {X 0,Y 361.978,Z 182.397,A -85,B 0,C 180,E1 -13153.899,E2 -13153.899} C_VEL
LIN {X 0,Y 361.95,Z 182.399,A -85,B 0,C 180,E1 -13157.94,E2 -13157.94} C_VEL
LIN {X 0,Y 361.874,Z 182.41,A -85,B 0,C 180,E1 -13161.654,E2 -13161.654} C_VEL
LIN {X 0,Y 361.911,Z 182.406,A -85,B 0,C 180,E1 -13165.292,E2 -13165.292} C_VEL
LIN {X 0,Y 361.903,Z 182.403,A -85,B 0,C 180,E1 -13167.78,E2 -13167.78} C_VEL
LIN {X 0,Y 361.833,Z 182.415,A -85,B 0,C 180,E1 -13171.287,E2 -13171.287} C_VEL
LIN {X 0,Y 361.841,Z 182.41,A -85,B 0,C 180,E1 -13174.282,E2 -13174.282} C_VEL
LIN {X 0,Y 361.85,Z 182.412,A -85,B 0,C 180,E1 -13177.224,E2 -13177.224} C_VEL
LIN {X 0,Y 361.824,Z 182.416,A -85,B 0,C 180,E1 -13180.757,E2 -13180.757} C_VEL
LIN {X 0,Y 361.807,Z 182.416,A -85,B 0,C 180,E1 -13184.371,E2 -13184.371} C_VEL
LIN {X 0,Y 361.824,Z 182.412,A -85,B 0,C 180,E1 -13187.571,E2 -13187.571} C_VEL
LIN {X 0,Y 361.818,Z 182.47,A -85,B 0,C 180,E1 -13190.984,E2 -13190.984} C_VEL
LIN {X 0,Y 361.888,Z 184.573,A -85,B 0,C 180,E1 -13192.987,E2 -13192.987} C_VEL
LIN {X 0,Y 361.754,Z 187.565,A -85,B 0,C 180,E1 -13195.711,E2 -13195.711} C_VEL
LIN {X 0,Y 361.462,Z 192.007,A -85,B 0,C 180,E1 -13199.635,E2 -13199.635} C_VEL
LIN {X 0,Y 361.22,Z 196.617,A -85,B 0,C 180,E1 -13203.508,E2 -13203.508} C_VEL
LIN {X 0,Y 360.975,Z 201.379,A -85,B 0,C 180,E1 -13207.387,E2 -13207.387} C_VEL
LIN {X 0,Y 360.965,Z 201.841,A -85,B 0,C 180,E1 -13207.689,E2 -13207.689} C_VEL
LIN {X 0,Y 364.484,Z 214.823,A -85,B 0,C 180,E1 -13208.399,E2 -13208.399} C_VEL
LIN {X 0,Y 367.186,Z 227.423,A -85,B 0,C 180,E1 -13209.271,E2 -13209.271} C_VEL
LIN {X 0,Y 367.967,Z 232.293,A -85,B 0,C 180,E1 -13209.658,E2 -13209.658} C_VEL
LIN {X 0,Y 367.195,Z 243.676,A -85,B 0,C 180,E1 -13210.577,E2 -13210.577} C_VEL
LIN {X 0,Y 366.047,Z 254.485,A -85,B 0,C 180,E1 -13211.676,E2 -13211.676} C_VEL
LIN {X 0,Y 365.012,Z 264.28,A -85,B 0,C 180,E1 -13212.925,E2 -13212.925} C_VEL
LIN {X 0,Y 363.915,Z 273.181,A -85,B 0,C 180,E1 -13214.314,E2 -13214.314} C_VEL
LIN {X 0,Y 363,Z 280.28,A -85,B 0,C 180,E1 -13215.659,E2 -13215.659} C_VEL
LIN {X 0,Y 362.305,Z 287.724,A -85,B 0,C 180,E1 -13217.395,E2 -13217.395} C_VEL
LIN {X 0,Y 361.544,Z 292.586,A -85,B 0,C 180,E1 -13218.791,E2 -13218.791} C_VEL
LIN {X 0,Y 361.112,Z 297.301,A -85,B 0,C 180,E1 -13220.478,E2 -13220.478} C_VEL
LIN {X 0,Y 360.747,Z 300.907,A -85,B 0,C 180,E1 -13222.162,E2 -13222.162} C_VEL
LIN {X 0,Y 360.517,Z 303.49,A -85,B 0,C 180,E1 -13223.834,E2 -13223.834} C_VEL
LIN {X 0,Y 360.434,Z 305.161,A -85,B 0,C 180,E1 -13225.526,E2 -13225.526} C_VEL
LIN {X 0,Y 360.314,Z 306.002,A -85,B 0,C 180,E1 -13227.764,E2 -13227.764} C_VEL
LIN {X 0,Y 360.346,Z 305.807,A -85,B 0,C 180,E1 -13228.882,E2 -13228.882} C_VEL
LIN {X 0,Y 360.418,Z 304.25,A -85,B 0,C 180,E1 -13231.116,E2 -13231.116} C_VEL
LIN {X 0,Y 360.538,Z 302.89,A -85,B 0,C 180,E1 -13232.233,E2 -13232.233} C_VEL
LIN {X 0,Y 360.787,Z 300.021,A -85,B 0,C 180,E1 -13233.908,E2 -13233.908} C_VEL
LIN {X 0,Y 361.053,Z 296.138,A -85,B 0,C 180,E1 -13235.584,E2 -13235.584} C_VEL
LIN {X 0,Y 361.536,Z 291.35,A -85,B 0,C 180,E1 -13237.189,E2 -13237.189} C_VEL
LIN {X 0,Y 362.127,Z 284.833,A -85,B 0,C 180,E1 -13238.93,E2 -13238.93} C_VEL
LIN {X 0,Y 362.974,Z 276.951,A -85,B 0,C 180,E1 -13240.598,E2 -13240.598} C_VEL
LIN {X 0,Y 364.127,Z 267.145,A -85,B 0,C 180,E1 -13242.256,E2 -13242.256} C_VEL
LIN {X 0,Y 365.091,Z 256.878,A -85,B 0,C 180,E1 -13243.638,E2 -13243.638} C_VEL
LIN {X 0,Y 365.786,Z 248.136,A -85,B 0,C 180,E1 -13244.604,E2 -13244.604} C_VEL
LIN {X 0,Y 366.66,Z 239.104,A -85,B 0,C 180,E1 -13245.422,E2 -13245.422} C_VEL
LIN {X 0,Y 367.076,Z 230.757,A -85,B 0,C 180,E1 -13246.052,E2 -13246.052} C_VEL
LIN {X 0,Y 364.952,Z 218.686,A -85,B 0,C 180,E1 -13246.908,E2 -13246.908} C_VEL
LIN {X 0,Y 362.067,Z 206.272,A -85,B 0,C 180,E1 -13247.598,E2 -13247.598} C_VEL
LIN {X 0,Y 360.933,Z 201.671,A -85,B 0,C 180,E1 -13247.819,E2 -13247.819} C_VEL
LIN {X 0,Y 361.094,Z 196.814,A -85,B 0,C 180,E1 -13251.701,E2 -13251.701} C_VEL
LIN {X 0,Y 361.297,Z 192.38,A -85,B 0,C 180,E1 -13255.335,E2 -13255.335} C_VEL
LIN {X 0,Y 361.546,Z 187.988,A -85,B 0,C 180,E1 -13259.073,E2 -13259.073} C_VEL
LIN {X 0,Y 361.704,Z 185.097,A -85,B 0,C 180,E1 -13261.639,E2 -13261.639} C_VEL
LIN {X 0,Y 361.739,Z 183.223,A -85,B 0,C 180,E1 -13263.339,E2 -13263.339} C_VEL
LIN {X 0,Y 361.702,Z 182.432,A -85,B 0,C 180,E1 -13264.293,E2 -13264.293} C_VEL
LIN {X 0,Y 361.734,Z 182.426,A -85,B 0,C 180,E1 -13264.716,E2 -13264.716} C_VEL
LIN {X 0,Y 361.154,Z 182.5,A -85,B 0,C 180,E1 -13265.647,E2 -13265.647} C_VEL
LIN {X 0,Y 358.383,Z 182.85,A -85,B 0,C 180,E1 -13267.161,E2 -13267.161} C_VEL
LIN {X 0,Y 355.969,Z 183.151,A -85,B 0,C 180,E1 -13268.386,E2 -13268.386} C_VEL
LIN {X 0,Y 354.896,Z 183.281,A -85,B 0,C 180,E1 -13269.332,E2 -13269.332} C_VEL
LIN {X 0,Y 354.792,Z 183.291,A -85,B 0,C 180,E1 -13269.653,E2 -13269.653} C_VEL
LIN {X 0,Y 354.778,Z 183.291,A -85,B 0,C 180,E1 -13272.865,E2 -13272.865} C_VEL
LIN {X 0,Y 354.825,Z 183.283,A -85,B 0,C 180,E1 -13276.112,E2 -13276.112} C_VEL
LIN {X 0,Y 354.84,Z 183.287,A -85,B 0,C 180,E1 -13279.186,E2 -13279.186} C_VEL
LIN {X 0,Y 354.789,Z 183.289,A -85,B 0,C 180,E1 -13282.4,E2 -13282.4} C_VEL
LIN {X 0,Y 354.791,Z 183.293,A -85,B 0,C 180,E1 -13284.938,E2 -13284.938} C_VEL
LIN {X 0,Y 354.771,Z 183.292,A -85,B 0,C 180,E1 -13288.403,E2 -13288.403} C_VEL
LIN {X 0,Y 354.828,Z 183.283,A -85,B 0,C 180,E1 -13291.617,E2 -13291.617} C_VEL
LIN {X 0,Y 354.875,Z 183.279,A -85,B 0,C 180,E1 -13294.17,E2 -13294.17} C_VEL
LIN {X 0,Y 354.835,Z 183.283,A -85,B 0,C 180,E1 -13297.894,E2 -13297.894} C_VEL
LIN {X 0,Y 354.897,Z 183.276,A -85,B 0,C 180,E1 -13301.89,E2 -13301.89} C_VEL
LIN {X 0,Y 354.915,Z 183.276,A -85,B 0,C 180,E1 -13305.98,E2 -13305.98} C_VEL
LIN {X 0,Y 354.968,Z 183.268,A -85,B 0,C 180,E1 -13309.735,E2 -13309.735} C_VEL
LIN {X 0,Y 355.088,Z 183.257,A -85,B 0,C 180,E1 -13312.036,E2 -13312.036} C_VEL
LIN {X 0,Y 355.074,Z 183.255,A -85,B 0,C 180,E1 -13314.32,E2 -13314.32} C_VEL
LIN {X 0,Y 355.214,Z 183.24,A -85,B 0,C 180,E1 -13317.732,E2 -13317.732} C_VEL
LIN {X 0,Y 355.323,Z 183.225,A -85,B 0,C 180,E1 -13320,E2 -13320} C_VEL
LIN {X 0,Y 355.222,Z 183.235,A -85,B 0,C 180,E1 -13322.268,E2 -13322.268} C_VEL
LIN {X 0,Y 355.112,Z 183.248,A -85,B 0,C 180,E1 -13326.819,E2 -13326.819} C_VEL
LIN {X 0,Y 354.99,Z 183.265,A -85,B 0,C 180,E1 -13329.113,E2 -13329.113} C_VEL
LIN {X 0,Y 354.897,Z 183.275,A -85,B 0,C 180,E1 -13332.582,E2 -13332.582} C_VEL
LIN {X 0,Y 354.859,Z 183.279,A -85,B 0,C 180,E1 -13336.097,E2 -13336.097} C_VEL
